Yaskawa INFORM job: SKRZYNIA_5340_-90_STOPNI_20BR.JBI

/JOB
//NAME SKRZYNIA_5340_-90_STOPNI_20BR
///FOLDERNAME 02-SKRZYNIE_JOBS
//POS
///NPOS 615,615,0,39,0,0
///TOOL 0
///POSTYPE PULSE
///PULSE
C00000=0,-52280,40443,0,6876,0
C00001=-82314,-24956,17040,-59626,-27382,-6248
C00002=-93910,-8625,17040,-59626,-43355,-6248
C00003=-98846,-1061,-42166,-80308,-57081,16120
C00004=-100452,6057,-48127,-85711,-56704,21322
C00005=-95817,31791,-34187,-84788,-63710,26674
C00006=-95573,33077,-33257,-84645,-64023,26851
C00007=-94315,33778,-32137,-85160,-63467,26714
C00008=-95573,33077,-33257,-84645,-64023,26851
C00009=-94948,31301,-36075,-85235,-63717,27152
C00010=-95573,33077,-33257,-84645,-64023,26851
C00011=-95263,33142,-33256,-84677,-63995,26850
C00012=-95263,33142,-33256,-84677,-63995,26850
C00013=-94230,33719,-32331,-85099,-63538,26735
C00014=-95263,33142,-33256,-84677,-63995,26850
C00015=-94794,31816,-35365,-85120,-63763,27076
C00016=-95263,33142,-33256,-84677,-63995,26850
C00017=-95260,33144,-33256,-84678,-63995,26850
C00018=-95260,33144,-33256,-84678,-63995,26850
C00019=-94260,33701,-32361,-85086,-63552,26738
C00020=-95260,33144,-33256,-84678,-63995,26850
C00021=-94835,31943,-35167,-85080,-63786,27056
C00022=-95260,33144,-33256,-84678,-63995,26850
C00023=-95258,25631,32269,-66559,-75499,2416
C00024=-95258,25631,32269,-66559,-75499,2416
C00025=-94256,26435,33444,-66420,-74940,2208
C00026=-95258,25631,32269,-66559,-75499,2416
C00027=-94857,24030,29962,-66606,-75105,2539
C00028=-95258,25631,32269,-66559,-75499,2416
C00029=-98811,21047,-15512,-99242,-81394,20987
C00030=-98811,21047,-15512,-99242,-81394,20987
C00031=-97856,21592,-14760,-99539,-80803,20995
C00032=-98811,21047,-15512,-99242,-81394,20987
C00033=-98487,19855,-17143,-99373,-81250,21110
C00034=-98811,21047,-15512,-99242,-81394,20987
C00035=-99077,36985,67047,-90824,-74996,11
C00036=-99077,36985,67047,-90824,-74996,11
C00037=-98126,38026,68808,-90519,-74354,-175
C00038=-99077,36985,67047,-90824,-74996,11
C00039=-98675,34279,62554,-90994,-74807,523
C00040=-99077,36985,67047,-90824,-74996,11
C00041=-98046,30065,45001,-99674,-75008,5996
C00042=-96663,27244,32711,-106417,-76052,10001
C00043=-96035,27733,33435,-106407,-75606,10011
C00044=-96663,27244,32711,-106417,-76052,10001
C00045=-96274,25568,30264,-106516,-75947,10234
C00046=-96663,27244,32711,-106417,-76052,10001
C00047=-93416,-2088,4699,-99676,-50441,9343
C00048=-88080,-20128,-3199,-80943,-31244,2335
C00049=-48287,-55439,-44481,-48508,-5390,-10469
C00050=-48287,-44591,-17414,-16172,-14532,-25809
C00051=-85348,-13130,13838,-41209,-47455,-8220
C00052=-97998,22495,32685,-69647,-75009,8900
C00053=-97362,30289,38867,-71738,-79704,10396
C00054=-97362,30289,38867,-71738,-79704,10396
C00055=-96447,31020,39967,-71637,-79179,10220
C00056=-97362,30289,38867,-71738,-79704,10396
C00057=-97069,28896,36765,-71776,-79401,10550
C00058=-97362,30289,38867,-71738,-79704,10396
C00059=-99590,25338,21334,-81459,-78469,-3358
C00060=-99590,25338,21334,-81459,-78469,-3358
C00061=-98681,25943,22203,-81468,-77867,-3455
C00062=-99590,25338,21334,-81459,-78469,-3358
C00063=-99296,24016,19444,-81525,-78239,-3225
C00064=-99590,25338,21334,-81459,-78469,-3358
C00065=-99820,26032,21623,-82067,-78848,-4447
C00066=-99820,26032,21623,-82067,-78848,-4447
C00067=-98898,26645,22513,-82083,-78237,-4546
C00068=-99820,26032,21623,-82067,-78848,-4447
C00069=-99438,24292,19129,-82156,-78552,-4268
C00070=-99820,26032,21623,-82067,-78848,-4447
C00071=-95331,1432,-9864,-84798,-60031,-3557
C00072=-95107,2197,-5510,-96695,-61306,-2364
C00073=-99461,26071,27151,-92834,-78756,-5773
C00074=-99144,26285,27462,-92832,-78536,-5787
C00075=-98121,27001,28507,-92822,-77820,-5838
C00076=-99144,26285,27462,-92832,-78536,-5787
C00077=-98815,24779,25284,-92901,-78347,-5607
C00078=-99144,26285,27462,-92832,-78536,-5787
C00079=-91210,-11403,-27677,-113165,-52408,5733
C00080=-98271,-15326,-41207,-114268,-59488,7673
C00081=-83743,-25164,-57719,-138536,-50905,17366
C00082=-83743,-25361,-52011,-136459,-47698,15842
C00083=-93071,-30029,-62286,-132724,-54351,14554
C00084=-61872,-66272,-83954,-148251,-32298,21081
C00085=-61872,-49557,-32264,-110357,-15428,1928
C00086=-65143,-26385,24751,-20080,-56896,-30933
C00087=-94996,555,46629,-41386,-61308,-21898
C00088=-98483,-26598,-36123,-71694,-41449,-2503
C00089=-98197,-8670,-25604,-81540,-55001,4479
C00090=-99236,18416,3235,-80713,-73731,6125
C00091=-98716,22747,8680,-80557,-75862,6048
C00092=-97982,23215,9333,-80619,-75386,5974
C00093=-98716,22747,8680,-80557,-75862,6048
C00094=-98409,21490,6932,-80649,-75627,6156
C00095=-98716,22747,8680,-80557,-75862,6048
C00096=-91715,3355,37300,-53415,-58440,-15905
C00097=-100183,29342,35466,-85708,-79719,1114
C00098=-100183,29342,35466,-85708,-79719,1114
C00099=-99011,30198,36753,-85631,-78926,990
C00100=-100183,29342,35466,-85708,-79719,1114
C00101=-99817,27493,32713,-85776,-79458,1347
C00102=-100183,29342,35466,-85708,-79719,1114
C00103=-99593,21150,23680,-85914,-74803,1967
C00104=-99593,30181,53843,-82632,-75568,-4688
C00105=-99618,36376,62891,-83676,-78551,-5246
C00106=-98461,37549,64848,-83362,-77827,-5489
C00107=-99618,36376,62891,-83676,-78551,-5246
C00108=-99260,34032,59054,-83761,-78261,-4840
C00109=-99618,36376,62891,-83676,-78551,-5246
C00110=-94729,-288,3800,-87543,-55904,1533
C00111=-77861,-26606,-19905,-76223,-21443,-3330
C00112=-46440,-50562,-32626,1826,-13880,-39178
C00113=-46440,-50562,-32626,1826,-13880,-39178
C00114=-38692,-65390,10180,-18335,3144,1955
C00115=0,-52280,40443,0,6876,0
C00116=0,-52280,40443,0,6876,0
C00117=0,-43112,23163,32261,-40956,29092
C00118=-48283,-21883,28214,-25170,-26491,48363
C00119=-46664,-3144,58041,-18842,-32105,45325
C00120=-50347,-18571,12268,-49104,-16423,60029
C00121=-52476,-17044,12146,-55476,-16783,62883
C00122=-51467,-16091,12918,-54586,-16145,62570
C00123=-51762,-16375,12685,-54854,-16332,62665
C00124=-53129,-15664,13268,-57063,-16995,63582
C00125=-52557,-17119,12084,-55547,-16837,62908
C00126=-52557,-17119,12084,-55547,-16837,62908
C00127=-52367,-16944,12224,-55385,-16717,62852
C00128=-50800,-15431,13458,-53958,-15729,62345
C00129=-51041,-15672,13259,-54187,-15881,62428
C00130=-52118,-15296,13570,-55899,-16415,63135
C00131=-51917,-16522,12564,-54988,-16433,62714
C00132=-50509,-19000,10610,-51503,-15997,61182
C00133=-52966,-16930,12240,-56194,-17032,63176
C00134=-51879,-15912,13067,-55265,-16346,62852
C00135=-52154,-16175,12851,-55507,-16521,62938
C00136=-53227,-15612,13314,-57215,-17042,63646
C00137=-52966,-16930,12240,-56194,-17032,63176
C00138=-50703,-18403,11066,-52155,-16024,61477
C00139=-52780,-17619,11680,-55562,-17015,62889
C00140=-51306,-16241,12790,-54268,-16084,62435
C00141=-51660,-16583,12512,-54593,-16308,62551
C00142=-53327,-15718,13220,-57282,-17114,63667
C00143=-52780,-17619,11680,-55562,-17015,62889
C00144=-50704,-18401,11069,-52157,-16021,61478
C00145=-53191,-17342,11901,-56260,-17204,63181
C00146=-51773,-16022,12969,-55050,-16305,62760
C00147=-52146,-16378,12679,-55379,-16540,62876
C00148=-53214,-15820,13135,-57085,-17059,63584
C00149=-53002,-17172,12037,-56105,-17083,63128
C00150=-51005,-17995,11387,-52847,-16122,61778
C00151=-52654,-17319,11922,-55560,-16911,62904
C00152=-51372,-16113,12897,-54432,-16099,62508
C00153=-51648,-16379,12679,-54684,-16273,62598
C00154=-52952,-15703,13233,-56807,-16903,63480
C00155=-53323,-17134,12070,-56539,-17248,63304
C00156=-52826,-20105,4812,-63938,-15678,66983
C00157=-52298,-19620,5183,-63681,-15322,66914
C00158=-51076,-18450,6096,-63049,-14499,66733
C00159=-51419,-18785,5831,-63233,-14731,66786
C00160=-52680,-18133,6347,-65138,-15424,67581
C00161=-52924,-19431,7025,-60935,-16175,65505
C00162=-51752,-18759,10786,-53484,-16613,62002
C00163=-52244,-17884,11471,-54682,-16766,62529
C00164=-50303,-16031,12961,-52880,-15542,61887
C00165=-50741,-16464,12607,-53310,-15818,62044
C00166=-52416,-15612,13306,-56135,-16617,63223
C00167=-51898,-18011,11369,-54129,-16600,62301
C00168=-50945,-18019,11363,-52741,-16103,61737
C00169=-51347,-17395,11856,-53690,-16237,62152
C00170=-49990,-16073,12923,-52376,-15383,61677
C00171=-50384,-16465,12603,-52769,-15629,61822
C00172=-52066,-15616,13298,-55654,-16423,63028
C00173=-51792,-17610,11685,-54205,-16494,62350
C00174=-50945,-18019,11363,-52741,-16103,61737
C00175=-50845,-17493,11778,-52895,-15987,61824
C00176=-49521,-16191,12826,-51571,-15155,61341
C00177=-49894,-16567,12520,-51958,-15389,61484
C00178=-51728,-15654,13268,-55171,-16246,62832
C00179=-51082,-17431,11827,-53280,-16102,61986
C00180=-50028,-23690,-6096,-22921,-31075,54538
C00181=-50346,-22995,-5584,-23393,-31002,54768
C00182=-48843,-21430,-4410,-21901,-30270,54078
C00183=-49178,-21788,-4683,-22239,-30433,54235
C00184=-50538,-21100,-4158,-23908,-30654,55032
C00185=-50252,-22811,-5450,-23315,-30936,54734
C00186=-49763,-24818,-32918,-23163,-28604,59699
C00187=-49144,-24298,-32242,-22455,-28505,59304
C00188=-47766,-22458,-30816,-21237,-27774,58615
C00189=-48099,-22913,-31171,-21534,-27949,58786
C00190=-49602,-21997,-30448,-23301,-28174,59772
C00191=-49259,-23869,-32392,-22880,-28141,59533
C00192=-50713,-12366,-58367,-41124,-17813,74400
C00193=-50097,-11438,-57505,-40749,-17495,74109
C00194=-49105,-9842,-55994,-40096,-16991,73614
C00195=-49355,-10250,-56383,-40269,-17116,73742
C00196=-50506,-9357,-55529,-41571,-17503,74586
C00197=-49771,-10920,-57018,-40545,-17327,73951
C00198=-46548,-30139,-39639,-20061,-27197,57955
C00199=-48797,-26670,-6576,-20404,-32539,53259
C00200=-45389,-28224,4312,-35967,-15579,54278
C00201=-40154,-51179,-915,-24203,-8234,36524
C00202=0,-52280,40443,0,6876,0
C00203=0,-52280,40443,0,6876,0
C00204=-2117,-50103,-33543,-4117,45077,85249
C00205=26439,-48928,-33543,-4117,-52362,85249
C00206=26439,-27355,-33543,-41485,-52362,85249
C00207=39218,-24492,-41653,-51934,-39374,86964
C00208=38244,-2284,-24157,-56964,-37300,90090
C00209=26640,586,-20198,-77712,-51919,89712
C00210=26323,460,-20341,-77681,-52125,89737
C00211=25607,3186,-17293,-77585,-52601,89760
C00212=26323,460,-20341,-77681,-52125,89737
C00213=27719,1044,-19697,-77798,-51218,89644
C00214=26640,586,-20198,-77712,-51919,89712
C00215=46457,7101,-11330,-26648,-40775,82885
C00216=47439,8350,-9833,-26106,-40556,82449
C00217=46334,10684,-6981,-26557,-41070,82837
C00218=47439,8350,-9833,-26106,-40556,82449
C00219=48354,9159,-8854,-25603,-40343,82046
C00220=47439,8350,-9833,-26106,-40556,82449
C00221=24760,-3019,-10726,-94610,-54398,89614
C00222=25145,-1220,-8811,-94681,-54143,89655
C00223=24492,1290,-6066,-94601,-54582,89624
C00224=25145,-1220,-8811,-94681,-54143,89655
C00225=26584,-669,-8211,-94866,-53174,89734
C00226=25145,-1220,-8811,-94681,-54143,89655
C00227=14532,-15164,-22494,-92943,-61192,88617
C00228=-33377,-12679,-20251,-90012,-93751,87621
C00229=-32674,-7309,22058,-70557,-98373,80594
C00230=20046,-29908,-41690,-58842,-55822,75080
C00231=46158,10269,-6164,-23128,-46470,70172
C00232=51306,10256,-19432,-23475,-33025,71236
C00233=50386,12004,-17260,-23922,-33430,71616
C00234=51306,10256,-19432,-23475,-33025,71236
C00235=51995,10928,-18601,-23012,-32906,70879
C00236=51306,10256,-19432,-23475,-33025,71236
C00237=50667,8104,-22050,-23976,-33027,71608
C00238=27434,3323,14960,-56922,-57501,78346
C00239=29014,6574,18756,-56344,-56678,77965
C00240=28326,9009,21700,-56459,-57175,78009
C00241=29014,6574,18756,-56344,-56678,77965
C00242=30292,7183,19486,-55908,-55969,77693
C00243=29014,6574,18756,-56344,-56678,77965
C00244=24457,-1296,-8898,-94600,-54606,89622
C00245=24457,-1296,-8898,-94600,-54606,89622
C00246=23939,748,-6672,-94541,-54956,89598
C00247=24457,-1296,-8898,-94600,-54606,89622
C00248=25626,-864,-8432,-94748,-53818,89684
C00249=24457,-1296,-8898,-94600,-54606,89622
C00250=22058,-20035,-26567,-93333,-56013,88551
C00251=-28907,-25632,-31027,-90338,-90583,86609
C00252=-23923,-11573,-19230,-90501,-87328,87840
C00253=-8646,-8251,-7782,-76032,-82054,83740
C00254=42001,26537,64712,-25019,-74648,68382
C00255=42692,25604,59505,-25067,-71864,68798
C00256=42100,27723,62792,-25233,-72628,68820
C00257=42692,25604,59505,-25067,-71864,68798
C00258=43179,26157,60355,-24838,-71882,68629
C00259=42692,25604,59505,-25067,-71864,68798
C00260=42064,17796,48100,-25604,-70267,69397
C00261=28113,-7386,-15136,-95790,-47335,90009
C00262=28228,-6488,-14240,-95859,-47266,90053
C00263=27767,-5044,-12775,-95858,-47588,90072
C00264=28228,-6488,-14240,-95859,-47266,90053
C00265=29468,-5989,-13737,-96077,-46438,90154
C00266=28228,-6488,-14240,-95859,-47266,90053
C00267=51937,664,-7429,-160484,-50080,89770
C00268=52345,1107,-6938,-160727,-50007,89930
C00269=51359,2767,-5080,-160136,-50147,89540
C00270=52345,1107,-6938,-160727,-50007,89930
C00271=53054,1752,-6222,-161147,-49882,90209
C00272=52345,1107,-6938,-160727,-50007,89930
C00273=51937,664,-7429,-160484,-50080,89770
C00274=29691,-10745,-18393,-95770,-46230,89933
C00275=26663,-19279,-25970,-94307,-48104,89008
C00276=29542,-7588,-14846,-100915,-46930,90773
C00277=29616,-6902,-10165,-96183,-45225,84004
C00278=29097,-5391,-8640,-96201,-45588,84023
C00279=29616,-6902,-10165,-96183,-45225,84004
C00280=31098,-6282,-9543,-96410,-44233,84135
C00281=29616,-6902,-10165,-96183,-45225,84004
C00282=7576,-30273,-44451,-97512,-61182,86443
C00283=-18624,-40022,-50597,-93591,-78329,83668
C00284=-32134,-30783,-37092,-96173,-88064,83581
C00285=23774,-1324,-8929,-94512,-55065,89585
C00286=23774,-1324,-8929,-94512,-55065,89585
C00287=23319,517,-6924,-94461,-55372,89567
C00288=23774,-1324,-8929,-94512,-55065,89585
C00289=25077,-853,-8421,-94674,-54188,89653
C00290=23774,-1324,-8929,-94512,-55065,89585
C00291=22107,-1052,28039,-94807,-51389,77849
C00292=19995,-16885,24938,-75612,-39910,62837
C00293=8393,-42921,36369,-24238,-5473,19544
C00294=0,-52280,40443,0,6876,0
C00295=-82314,-24956,17040,-59626,-27382,-6248
C00296=-93910,-8625,17040,-59626,-43355,-6248
C00297=-98846,-1061,-42166,-80308,-57081,16120
C00298=-100452,6057,-48127,-85711,-56704,21322
C00299=-95564,34698,-34234,-85516,-63941,27819
C00300=-94021,36658,-30981,-84167,-64832,27454
C00301=-93851,36773,-30815,-84181,-64812,27439
C00302=-95564,34698,-34234,-85516,-63941,27819
C00303=-96930,32282,-32252,-82595,-65816,26305
C00304=-93901,32995,-31122,-83953,-64436,26132
C00305=-93891,32978,-31150,-83961,-64431,26134
C00306=-96930,32282,-32252,-82595,-65816,26305
C00307=-97719,-4194,-31542,-76086,-54596,10626
C00308=-88377,-34186,-45291,-67238,-52212,2442
C00309=-73560,-62084,7826,-28695,-34737,-3666
C00310=0,-52280,40443,0,6876,0
C00311=0,-52280,40443,0,6876,0
C00312=-2117,-50103,-33543,-4117,45077,85249
C00313=26439,-48928,-33543,-4117,-52362,85249
C00314=26439,-27355,-33543,-41485,-52362,85249
C00315=39218,-24492,-41653,-51934,-39374,86964
C00316=37381,-5106,-22608,-53943,-39515,88347
C00317=38119,-10689,-19379,-70548,-34101,88029
C00318=37906,-14512,-22901,-69984,-34376,87713
C00319=41414,6981,-5927,-33889,-45598,86373
C00320=42289,10624,-1511,-33365,-45508,85956
C00321=42351,10656,-1473,-33340,-45486,85935
C00322=41414,6981,-5927,-33889,-45598,86373
C00323=53221,-12364,-8957,-19277,-47766,73858
C00324=11365,-15171,10010,-30164,-77975,82960
C00325=16156,-38280,11293,-23671,-42998,42040
C00326=11365,-47379,10010,-30164,3063,681
C00327=0,-52280,40443,0,6876,0
C00328=0,-36700,24612,42871,-31823,33862
C00329=-44403,-30110,7154,-24155,-23805,45557
C00330=-51570,-19542,10947,-41619,-21811,53396
C00331=-51570,-17239,16856,-38066,-23574,51584
C00332=-55052,-13712,19754,-43494,-24529,53873
C00333=-55190,-12778,21730,-42693,-25060,53437
C00334=-40431,-28773,9158,-17648,-23273,42875
C00335=0,-36700,24612,42871,-31823,33862
C00336=0,-52280,40443,0,6876,0
C00337=0,-52280,40443,0,6876,0
C00338=-73560,-62084,7826,-28695,-34737,-3666
C00339=-88377,-34186,-45291,-67238,-52212,2442
C00340=-99860,-8392,-35780,-75647,-56000,10650
C00341=-100432,21324,12575,-83706,-77956,7498
C00342=-100432,21324,12575,-83706,-77956,7498
C00343=-97477,24790,17443,-83584,-77881,7143
C00344=-97548,25214,18044,-83537,-78171,7107
C00345=-100432,21324,12575,-83706,-77956,7498
C00346=-100473,21504,12824,-83696,-77986,7482
C00347=-97708,25565,18549,-83502,-78342,7077
C00348=-97720,26100,19317,-83456,-78605,7025
C00349=-100432,21324,12575,-83706,-77956,7498
C00350=-98403,3681,-8965,-86029,-63956,7946
C00351=-98851,2841,7216,-80537,-62817,1838
C00352=-99868,-33,22146,-72719,-59601,-5126
C00353=-99028,-10516,17309,-71061,-60695,-4227
C00354=-58820,-39124,10926,-53325,-41870,-3759
C00355=0,-52280,40443,0,6876,0
C00356=-37281,-50778,-9546,-79570,-75313,71156
C00357=-21038,-23698,-30323,-82948,-81132,85647
C00358=-21230,-24252,-33397,-84866,-81311,86227
C00359=26224,-11477,-22521,-89106,-49066,87170
C00360=30473,789,4724,-68168,-47848,79016
C00361=30460,-1091,-3608,-71823,-46530,81583
C00362=26224,-11477,-22521,-89106,-49066,87170
C00363=1250,-26379,-34995,-85812,-66036,85728
C00364=-29373,-17697,-13794,-84248,-87305,82376
C00365=-12562,-22815,-22029,-52123,-75138,85349
C00366=41964,2536,-13642,-34848,-42769,74522
C00367=37974,4101,-26304,-58477,-36842,84551
C00368=37992,4823,-31618,-63468,-34913,87461
C00369=41439,5489,-14791,-37032,-40569,75962
C00370=38833,-3286,10682,-41231,-51577,69207
C00371=-9276,-22918,-17698,-90837,-69000,78700
C00372=-8172,-56778,-49528,-75726,-40055,75711
C00373=-3982,-61001,-53003,-69042,-33087,73336
C00374=37287,-55159,35520,-2191,5667,2084
C00375=0,-52280,40443,0,6876,0
C00376=0,-36700,24612,42871,-31823,33862
C00377=-44403,-30110,7154,-24155,-23805,45557
C00378=-44403,-30110,7154,-24155,-23805,45557
C00379=-42101,-12213,25656,-103795,-5192,78630
C00380=-46259,-8171,27719,-110365,-8144,81138
C00381=-49067,-3914,32085,-108223,-9817,79727
C00382=-55938,-2414,24284,-132193,-25662,89374
C00383=-55195,18277,75263,-85826,-17009,66357
C00384=-37783,26295,96734,15514,-13481,23189
C00385=-56934,-15752,2926,-132390,-27589,90381
C00386=-47073,-34549,9488,-27883,-30316,51458
C00387=0,-52280,40443,0,6876,0
C00388=0,-52280,40443,0,6876,0
C00389=-73560,-62084,7826,-28695,-34737,-3666
C00390=-96366,-17217,16860,-56620,-71703,-18245
C00391=-98152,-14905,2044,-65675,-67485,-3494
C00392=-100467,-7393,-15195,-81625,-60158,6002
C00393=-99336,18440,8642,-84276,-74234,7647
C00394=-99336,18440,8642,-84276,-74234,7647
C00395=-97907,25479,18429,-83510,-78268,7080
C00396=-97774,25771,18838,-83486,-78362,7054
C00397=-99336,18440,8642,-84276,-74234,7647
C00398=-99336,20364,19482,-82786,-74642,4774
C00399=-98337,25059,18813,-87846,-78771,10707
C00400=-98337,23926,10585,-88652,-78855,12971
C00401=-99528,19847,13673,-83665,-74506,6500
C00402=-89817,-17341,-38408,-97132,-45323,12250
C00403=-100347,-21961,-42251,-93939,-52125,11121
C00404=-60204,-59872,-73451,-117647,-17639,18840
C00405=-37721,-67612,11381,-1325,-438,-7850
C00406=0,-52280,40443,0,6876,0
C00407=37287,-55159,35520,-2191,5667,2084
C00408=40042,-68802,-18337,-47708,-19461,45384
C00409=16481,-63411,-38742,-86271,-37962,67106
C00410=28646,-23138,-32952,-89786,-42552,85395
C00411=38882,-16596,-17625,-44304,-41043,72768
C00412=40930,-6862,-13364,-47045,-37020,74415
C00413=41744,-3361,-9781,-46774,-36492,74231
C00414=41678,-4243,-16493,-50979,-33997,76666
C00415=40930,-6862,-13364,-47045,-37020,74415
C00416=38882,-16596,-17625,-44304,-41043,72768
C00417=28646,-23138,-32952,-89786,-42552,85395
C00418=29905,-15291,-26411,-91102,-43435,86304
C00419=31540,-7654,-19248,-92177,-42391,86919
C00420=31445,-8095,-22888,-97196,-43117,89457
C00421=29637,-16450,-35189,-96198,-44206,89682
C00422=-7164,-46429,-55577,-86274,-68578,84143
C00423=40042,-68802,-18337,-47708,-19461,45384
C00424=37287,-55159,35520,-2191,5667,2084
C00425=0,-52280,40443,0,6876,0
C00426=-37164,-60659,6466,-13301,-5027,19773
C00427=-45362,-39990,2831,-27538,-17767,40935
C00428=-57189,-26834,-7130,-38780,-31731,51561
C00429=-55974,-20661,-3180,-39617,-29741,52134
C00430=-55991,-28453,-45977,-64163,-20900,63765
C00431=-57189,-26834,-7130,-38780,-31731,51561
C00432=-41180,-61187,4729,-17280,-8498,23442
C00433=0,-52280,40443,0,6876,0
C00434=0,-52280,40443,0,6876,0
C00435=-43180,-50572,-20637,-6552,-29302,-38834
C00436=-79425,-37128,-15462,-51820,-35721,-18807
C00437=-93702,-21743,-5664,-65079,-41536,-12324
C00438=-94876,-11469,-23586,-124528,-59237,5423
C00439=-92861,23404,17376,-116518,-76732,-1573
C00440=-91304,28381,24747,-115873,-78046,-2652
C00441=-91460,31648,35777,-114879,-76291,-4970
C00442=-92889,23503,17516,-116511,-76737,-1586
C00443=-94876,-11469,-23586,-124528,-59237,5423
C00444=-94108,-26192,-19530,-80749,-38523,-6311
C00445=-79425,-37128,-15462,-51820,-35721,-18807
C00446=-44920,-50063,-20090,-8739,-29356,-37564
C00447=-37721,-67612,11381,-1325,-438,-7850
C00448=0,-52280,40443,0,6876,0
C00449=40043,-68802,-18337,-47706,-19461,45383
C00450=27078,-46675,7729,-35821,-60236,53359
C00451=37661,6027,34279,-36092,-58837,68690
C00452=38848,9668,32452,-36978,-55195,69693
C00453=45203,15557,41040,-24527,-60177,66840
C00454=37661,2340,23735,-37788,-55306,70200
C00455=22173,-30639,7984,-58136,-45615,60133
C00456=37287,-55159,35520,-2191,5667,2084
C00457=0,-52280,40443,0,6876,0
C00458=-23708,-46776,23536,-16027,-4787,19738
C00459=-50917,-40459,4132,-34421,-18173,42391
C00460=-54964,-26842,8528,-44141,-23181,52038
C00461=-51719,-20944,8196,-48593,-18539,54728
C00462=-53338,-16066,12564,-52314,-18938,56375
C00463=-53668,-14237,17353,-48629,-20286,54493
C00464=-18010,-41727,-5437,24633,-20435,23511
C00465=-41180,-61187,4729,-17280,-8498,23442
C00466=0,-52280,40443,0,6876,0
C00467=0,-52280,40443,0,6876,0
C00468=-37721,-67612,11381,-1325,-438,-7850
C00469=-43180,-50572,-20637,-6552,-29302,-38834
C00470=-79425,-37128,-15462,-51820,-35721,-18807
C00471=-92377,-33385,-41303,-83059,-36844,-1354
C00472=-98996,-8012,-20669,-89286,-58253,3196
C00473=-99186,-1007,-13605,-90357,-63007,3800
C00474=-99448,23410,16807,-87478,-77479,2357
C00475=-98529,24761,18725,-87324,-78429,2215
C00476=-98419,25196,20150,-87169,-78534,1864
C00477=-99450,-173,-12700,-90327,-63185,3798
C00478=-99875,3426,-9244,-98609,-66692,6315
C00479=-99431,-3293,-16601,-99643,-62713,6757
C00480=-92822,-26306,-37175,-103295,-43881,7703
C00481=-68601,-52593,-52127,-95725,-25602,3235
C00482=-80632,-38079,-20908,-64053,-45216,-12949
C00483=-43180,-50572,-20637,-6552,-29302,-38834
C00484=-37721,-67612,11381,-1325,-438,-7850
C00485=0,-52280,40443,0,6876,0
C00486=-7830,-25136,17099,-55306,-64068,52084
C00487=34592,-23156,18291,-29932,-45204,43222
C00488=27626,-5609,7480,-74303,-46810,69713
C00489=30162,-7263,-3756,-79871,-43922,73611
C00490=30945,-3557,12,-79972,-43367,73694
C00491=30934,-3652,-86,-79966,-43372,73693
C00492=29106,-7674,-4162,-79972,-44640,73655
C00493=-2837,-32019,-23857,-80741,-66785,72567
C00494=9534,-43450,13514,-26959,-29486,38723
C00495=22834,-59963,22946,-6692,-2150,9612
C00496=0,-52280,40443,0,6876,0
C00497=-23708,-46776,23536,-16027,-4787,19738
C00498=-50917,-40459,4132,-34421,-18173,42391
C00499=-51059,-36587,4608,-36647,-19418,45358
C00500=-50113,-22729,10834,-36393,-23396,50963
C00501=-58003,-17258,7975,-66354,-22196,69294
C00502=-57660,-15851,11780,-61832,-22634,66694
C00503=-50113,-22729,10834,-36393,-23396,50963
C00504=-45969,-44671,-42317,80322,10570,10889
C00505=-31285,-69981,-10849,-7246,-6842,20992
C00506=0,-52280,40443,0,6876,0
C00507=-37721,-67612,11381,-1325,-438,-7850
C00508=-43180,-50572,-20637,-6552,-29302,-38834
C00509=-79425,-37128,-15462,-51820,-35721,-18807
C00510=-92377,-33385,-41303,-83059,-36844,-1354
C00511=-97955,-4566,-17156,-86109,-58691,2381
C00512=-98023,-4368,-16953,-86108,-58737,2386
C00513=-97622,-3602,-16155,-86160,-58465,2400
C00514=-99754,24347,18348,-83049,-78046,1543
C00515=-98401,23935,17754,-83131,-77323,1564
C00516=-98274,24050,17917,-83129,-77329,1551
C00517=-99954,24418,19993,-82828,-78557,1051
C00518=-99712,24798,18984,-83012,-78332,1506
C00519=-99852,25442,19906,-82977,-78439,1439
C00520=-98294,26390,21274,-82926,-78604,1336
C00521=-98320,27540,23370,-82787,-79202,1083
C00522=-100298,21581,9800,-87114,-77804,3862
C00523=-100167,24076,23961,-91830,-78070,1153
C00524=-97934,23655,23660,-91877,-76543,1161
C00525=-97934,26645,35668,-90599,-76116,-1688
C00526=-100333,13965,-3660,-96424,-75767,7039
C00527=-99852,25442,19906,-82977,-78439,1439
C00528=-99768,8894,-2445,-89351,-68751,3793
C00529=-96099,-3787,-16815,-92200,-58195,4535
C00530=-97559,-25159,-36085,-93407,-46496,3918
C00531=-68601,-52593,-52127,-95725,-25602,3235
C00532=-80632,-38079,-20908,-64053,-45216,-12949
C00533=-43180,-50572,-20637,-6552,-29302,-38834
C00534=-37721,-67612,11381,-1325,-438,-7850
C00535=54026,-30203,28811,7745,-28969,5087
C00536=55906,-29650,27841,6704,-28568,42061
C00537=3910,-49110,-20873,-64325,-51391,71742
C00538=9596,-41005,-15480,-61992,-50741,70573
C00539=34629,-5327,8260,-51720,-47880,65426
C00540=35679,2837,17551,-51053,-47466,65038
C00541=35689,-56,7549,-54586,-44718,67469
C00542=34629,-5327,8260,-51720,-47880,65426
C00543=9596,-41005,-15480,-61992,-50741,70573
C00544=29660,-4584,-26917,-122917,-59269,85605
C00545=30458,-1431,-23593,-123278,-58903,85810
C00546=32051,-581,-21149,-126899,-58917,85995
C00547=28378,-5181,-30467,-124970,-61925,86269
C00548=9596,-41005,-15480,-61992,-50741,70573
C00549=4124,-42500,-16101,-63937,-54198,71061
C00550=22834,-59963,22946,-6692,-2150,9612
C00551=0,-52280,40443,0,6876,0
C00552=-44101,-76445,-48847,-15697,-17168,40457
C00553=-48984,-30078,-36716,-21434,-29637,58750
C00554=-50484,-13386,-55713,-36158,-19724,71897
C00555=-50319,-9878,-52358,-36554,-19395,72071
C00556=-57778,15231,-57159,-77377,-21293,89265
C00557=-50484,-13386,-55713,-36158,-19724,71897
C00558=-49763,-25421,-36239,-24565,-26935,60445
C00559=-50529,-22709,-3778,-22940,-31995,54502
C00560=-45389,-28224,4312,-35967,-15579,54278
C00561=-40154,-51179,-915,-24203,-8234,36524
C00562=0,-52280,40443,0,6876,0
C00563=0,-52280,40443,0,6876,0
C00564=-37721,-67612,11381,-1325,-438,-7850
C00565=-43180,-50572,-20637,-6552,-29302,-38834
C00566=-43180,-50572,-20637,-6552,-29302,-38834
C00567=-91571,-17240,10754,-52986,-45776,-17944
C00568=-95322,4002,18806,-71534,-58652,-8117
C00569=-84901,-1641,24348,-52361,-47087,-17020
C00570=-100018,24469,26124,-84922,-77496,-993
C00571=-98221,24171,26084,-84881,-76275,-1110
C00572=-97925,23780,23736,-81145,-76027,-1196
C00573=-96763,24072,23316,-74311,-75270,-2269
C00574=-95281,25990,27886,-68316,-75415,-4201
C00575=-99355,23812,23162,-76774,-76908,-1703
C00576=-99772,22813,18672,-85812,-76963,849
C00577=-98588,26860,21106,-87462,-79585,-1754
C00578=-98621,27173,20618,-87985,-79896,-2348
C00579=-99360,20896,24116,-84704,-74336,-1671
C00580=-99329,20456,17173,-93067,-75506,1686
C00581=-97621,19686,17216,-93018,-74287,1457
C00582=-97553,22128,27761,-91636,-73750,-1130
C00583=-97912,34558,59975,-88815,-75536,-7324
C00584=-97912,45071,86162,-86500,-75470,-12145
C00585=-89794,-9992,-7341,-81590,-44258,-3681
C00586=-98228,-14972,-11291,-81392,-49231,-4002
C00587=-98228,-7428,13566,-72439,-51372,-10695
C00588=-68865,-35989,-5252,-49829,-38105,-21179
C00589=-15566,-52364,-9989,12732,-35649,-46896
C00590=0,-52278,40443,-31822,-65283,46097
C00591=7820,3000,44222,-77356,-66876,70486
C00592=23103,22769,71034,-65639,-61603,67373
C00593=25078,30713,84198,-63240,-61811,65668
C00594=25008,30264,83410,-63369,-61766,65773
C00595=23103,22769,71034,-65639,-61603,67373
C00596=23103,22769,71034,-65639,-61603,67373
C00597=25078,30713,84198,-63240,-61811,65668
C00598=25008,30264,83410,-63369,-61766,65773
C00599=23103,22769,71034,-65639,-61603,67373
C00600=-3014,-20441,-7349,-104591,-68614,79454
C00601=-3014,-20441,-7349,-104591,-68614,79454
C00602=-13238,-21720,-1359,-93359,-59492,72612
C00603=10261,-46634,14475,-36899,-22136,31570
C00604=22834,-59963,22946,-6692,-2150,9612
C00605=0,-52280,40443,0,6876,0
C00606=-23708,-46776,23536,-16027,-4787,19738
C00607=-50917,-40459,4132,-34421,-18173,42391
C00608=-49876,-21948,7530,-68838,-10324,59148
C00609=-46721,-18942,9765,-68167,-8197,59205
C00610=-47734,-15041,12007,-78406,-8476,63945
C00611=-48173,-14749,12492,-78097,-8776,63748
C00612=-42573,-24036,4541,-56448,-5917,54155
C00613=-31287,-69981,-10850,-7253,-6843,20996
C00614=0,-52280,40443,0,6876,0
BC00000=455888
BC00001=445130
BC00002=445130
BC00003=445130
BC00004=445130
BC00005=467179
BC00006=468227
BC00007=468227
BC00008=468227
BC00009=468227
BC00010=468227
BC00011=514421
BC00012=514421
BC00013=514421
BC00014=514421
BC00015=514421
BC00016=514421
BC00017=560588
BC00018=560588
BC00019=560588
BC00020=560588
BC00021=560588
BC00022=560588
BC00023=536404
BC00024=536404
BC00025=536404
BC00026=536404
BC00027=536404
BC00028=536404
BC00029=582458
BC00030=582458
BC00031=582458
BC00032=582458
BC00033=582458
BC00034=582458
BC00035=581206
BC00036=581206
BC00037=581206
BC00038=581206
BC00039=581206
BC00040=581206
BC00041=608443
BC00042=626741
BC00043=626741
BC00044=626741
BC00045=626741
BC00046=626741
BC00047=604255
BC00048=604255
BC00049=627238
BC00050=699121
BC00051=714117
BC00052=772491
BC00053=770398
BC00054=770398
BC00055=770398
BC00056=770398
BC00057=770398
BC00058=770398
BC00059=820815
BC00060=820815
BC00061=820815
BC00062=820815
BC00063=820815
BC00064=820815
BC00065=866263
BC00066=866263
BC00067=866263
BC00068=866263
BC00069=866263
BC00070=866263
BC00071=866263
BC00072=904896
BC00073=904896
BC00074=904896
BC00075=904896
BC00076=904896
BC00077=904896
BC00078=904896
BC00079=872244
BC00080=872244
BC00081=872244
BC00082=872244
BC00083=872244
BC00084=872244
BC00085=872244
BC00086=943472
BC00087=944390
BC00088=976590
BC00089=976703
BC00090=960530
BC00091=953739
BC00092=953739
BC00093=953739
BC00094=953739
BC00095=953739
BC00096=949233
BC00097=963886
BC00098=963886
BC00099=963886
BC00100=963886
BC00101=963886
BC00102=963886
BC00103=963886
BC00104=1017492
BC00105=1017492
BC00106=1017492
BC00107=1017492
BC00108=1017492
BC00109=1017492
BC00110=969716
BC00111=953277
BC00112=956863
BC00113=935999
BC00114=860772
BC00115=811795
BC00116=811793
BC00117=811795
BC00118=919701
BC00119=919701
BC00120=949003
BC00121=953382
BC00122=953382
BC00123=953382
BC00124=953382
BC00125=953382
BC00126=1005542
BC00127=1006846
BC00128=1006846
BC00129=1006846
BC00130=1006846
BC00131=1006846
BC00132=888056
BC00133=888056
BC00134=888056
BC00135=888056
BC00136=888056
BC00137=888056
BC00138=830714
BC00139=830714
BC00140=830714
BC00141=830714
BC00142=830714
BC00143=830714
BC00144=764829
BC00145=764829
BC00146=764829
BC00147=764829
BC00148=764829
BC00149=764829
BC00150=707174
BC00151=707174
BC00152=707174
BC00153=707174
BC00154=707174
BC00155=707174
BC00156=642071
BC00157=642071
BC00158=642071
BC00159=642071
BC00160=642071
BC00161=642071
BC00162=584746
BC00163=584746
BC00164=584746
BC00165=584746
BC00166=584746
BC00167=584746
BC00168=519232
BC00169=519232
BC00170=519232
BC00171=519232
BC00172=519232
BC00173=519232
BC00174=461813
BC00175=461813
BC00176=461813
BC00177=461813
BC00178=461813
BC00179=461813
BC00180=459544
BC00181=459544
BC00182=459544
BC00183=459544
BC00184=459544
BC00185=459544
BC00186=459544
BC00187=459544
BC00188=459544
BC00189=459544
BC00190=459544
BC00191=459544
BC00192=459544
BC00193=459544
BC00194=459544
BC00195=459544
BC00196=459544
BC00197=459544
BC00198=459544
BC00199=459544
BC00200=459540
BC00201=533216
BC00202=533216
BC00203=492150
BC00204=423885
BC00205=423885
BC00206=423885
BC00207=423885
BC00208=423885
BC00209=423882
BC00210=423882
BC00211=423882
BC00212=423882
BC00213=423882
BC00214=423882
BC00215=517447
BC00216=516208
BC00217=516208
BC00218=516208
BC00219=516208
BC00220=516208
BC00221=462401
BC00222=462401
BC00223=462401
BC00224=462401
BC00225=462401
BC00226=462401
BC00227=462401
BC00228=462401
BC00229=581968
BC00230=647467
BC00231=647467
BC00232=647467
BC00233=647467
BC00234=647467
BC00235=647467
BC00236=647467
BC00237=647467
BC00238=600589
BC00239=600589
BC00240=600589
BC00241=600589
BC00242=600589
BC00243=600589
BC00244=646713
BC00245=646713
BC00246=646713
BC00247=646713
BC00248=646713
BC00249=646713
BC00250=646713
BC00251=646713
BC00252=703926
BC00253=764819
BC00254=734650
BC00255=734650
BC00256=734650
BC00257=734650
BC00258=734650
BC00259=734650
BC00260=734650
BC00261=762000
BC00262=762000
BC00263=762000
BC00264=762000
BC00265=762000
BC00266=762000
BC00267=768744
BC00268=768744
BC00269=768744
BC00270=768744
BC00271=768744
BC00272=768744
BC00273=768744
BC00274=762000
BC00275=762000
BC00276=869424
BC00277=869424
BC00278=869424
BC00279=869424
BC00280=869424
BC00281=869424
BC00282=869424
BC00283=869424
BC00284=983898
BC00285=992364
BC00286=992364
BC00287=992364
BC00288=992364
BC00289=992364
BC00290=992364
BC00291=927243
BC00292=910363
BC00293=791398
BC00294=458496
BC00295=445130
BC00296=445130
BC00297=445130
BC00298=445130
BC00299=475938
BC00300=475917
BC00301=468314
BC00302=475938
BC00303=515329
BC00304=515329
BC00305=508301
BC00306=515329
BC00307=542207
BC00308=542207
BC00309=542207
BC00310=542207
BC00311=492150
BC00312=423885
BC00313=423885
BC00314=423885
BC00315=423885
BC00316=418215
BC00317=406365
BC00318=406365
BC00319=507950
BC00320=507950
BC00321=500226
BC00322=507950
BC00323=493160
BC00324=493160
BC00325=493160
BC00326=493160
BC00327=493160
BC00328=582810
BC00329=655182
BC00330=714528
BC00331=712780
BC00332=712780
BC00333=773753
BC00334=773753
BC00335=582810
BC00336=540924
BC00337=542207
BC00338=542207
BC00339=542207
BC00340=590944
BC00341=543764
BC00342=459277
BC00343=459277
BC00344=451665
BC00345=459277
BC00346=520748
BC00347=520748
BC00348=528295
BC00349=520748
BC00350=524597
BC00351=612873
BC00352=584417
BC00353=584417
BC00354=584417
BC00355=584417
BC00356=542360
BC00357=599440
BC00358=482963
BC00359=482963
BC00360=482963
BC00361=482963
BC00362=482963
BC00363=482963
BC00364=482963
BC00365=633179
BC00366=633182
BC00367=633182
BC00368=633182
BC00369=633182
BC00370=590162
BC00371=577838
BC00372=565789
BC00373=612529
BC00374=620193
BC00375=620193
BC00376=812803
BC00377=887783
BC00378=927066
BC00379=893694
BC00380=914884
BC00381=914884
BC00382=943670
BC00383=952070
BC00384=963270
BC00385=945981
BC00386=853059
BC00387=542207
BC00388=542207
BC00389=513519
BC00390=556866
BC00391=576802
BC00392=590944
BC00393=571989
BC00394=566860
BC00395=566866
BC00396=572997
BC00397=566860
BC00398=625806
BC00399=632891
BC00400=631419
BC00401=627770
BC00402=635118
BC00403=635118
BC00404=633159
BC00405=733103
BC00406=733103
BC00407=620193
BC00408=620193
BC00409=625652
BC00410=635598
BC00411=635598
BC00412=635598
BC00413=635598
BC00414=635598
BC00415=635598
BC00416=635598
BC00417=635598
BC00418=658627
BC00419=658630
BC00420=665879
BC00421=658627
BC00422=658627
BC00423=620193
BC00424=620193
BC00425=620193
BC00426=561542
BC00427=498768
BC00428=452071
BC00429=452071
BC00430=452071
BC00431=452071
BC00432=524165
BC00433=524165
BC00434=733103
BC00435=733103
BC00436=615417
BC00437=615411
BC00438=615411
BC00439=615411
BC00440=615411
BC00441=615411
BC00442=615411
BC00443=615411
BC00444=615411
BC00445=615417
BC00446=698572
BC00447=733103
BC00448=733103
BC00449=667407
BC00450=721208
BC00451=721208
BC00452=721208
BC00453=727232
BC00454=730010
BC00455=686453
BC00456=620193
BC00457=620193
BC00458=576077
BC00459=541793
BC00460=580754
BC00461=589556
BC00462=589433
BC00463=647350
BC00464=649294
BC00465=561088
BC00466=547800
BC00467=733103
BC00468=733103
BC00469=733103
BC00470=733103
BC00471=757807
BC00472=750752
BC00473=747214
BC00474=740531
BC00475=740531
BC00476=745553
BC00477=740531
BC00478=750469
BC00479=750469
BC00480=750469
BC00481=750469
BC00482=783373
BC00483=795297
BC00484=733103
BC00485=733103
BC00486=727492
BC00487=727492
BC00488=759331
BC00489=759331
BC00490=759331
BC00491=766564
BC00492=759331
BC00493=759331
BC00494=672725
BC00495=672725
BC00496=672725
BC00497=766882
BC00498=791101
BC00499=802867
BC00500=836517
BC00501=836517
BC00502=895002
BC00503=836517
BC00504=798026
BC00505=767805
BC00506=733103
BC00507=733103
BC00508=733103
BC00509=733103
BC00510=768965
BC00511=777113
BC00512=815683
BC00513=817504
BC00514=817504
BC00515=817504
BC00516=824335
BC00517=824335
BC00518=862603
BC00519=862905
BC00520=863393
BC00521=870426
BC00522=870426
BC00523=904292
BC00524=904292
BC00525=904292
BC00526=904292
BC00527=862905
BC00528=824848
BC00529=818776
BC00530=812035
BC00531=750469
BC00532=783373
BC00533=795297
BC00534=733103
BC00535=762701
BC00536=765633
BC00537=830967
BC00538=835024
BC00539=852883
BC00540=852883
BC00541=852883
BC00542=852883
BC00543=835024
BC00544=861491
BC00545=861491
BC00546=861491
BC00547=861491
BC00548=835024
BC00549=835024
BC00550=672725
BC00551=672725
BC00552=528256
BC00553=459544
BC00554=459544
BC00555=459544
BC00556=459544
BC00557=459544
BC00558=459544
BC00559=459544
BC00560=459540
BC00561=533216
BC00562=533216
BC00563=733103
BC00564=733103
BC00565=854587
BC00566=967109
BC00567=948121
BC00568=961016
BC00569=923671
BC00570=946274
BC00571=946274
BC00572=946274
BC00573=946274
BC00574=946274
BC00575=946274
BC00576=970029
BC00577=970060
BC00578=977448
BC00579=970029
BC00580=1018114
BC00581=1018114
BC00582=1018114
BC00583=1018114
BC00584=1018114
BC00585=975782
BC00586=976838
BC00587=956699
BC00588=952322
BC00589=952322
BC00590=921533
BC00591=921533
BC00592=946591
BC00593=946591
BC00594=953713
BC00595=946591
BC00596=997282
BC00597=997282
BC00598=1004404
BC00599=997282
BC00600=1013986
BC00601=963295
BC00602=908449
BC00603=754884
BC00604=672725
BC00605=672725
BC00606=562340
BC00607=452362
BC00608=452362
BC00609=452362
BC00610=452362
BC00611=512870
BC00612=511886
BC00613=742282
BC00614=742282
///POSTYPE BASE
///RECTAN
///RCONF 1,0,0,0,0,0,0,0,0,0,0,0,0,0,0,0,0,0,0,0,0,0,0,0
P00006=0.000,0.000,0.000,0.0000,0.0000,0.0000
P00300=-0.036,-1.505,2.318,0.0000,0.0000,0.0000
P00301=0.046,-2.112,7.779,0.0000,0.0000,0.0000
P00302=-0.180,-2.409,6.326,0.0000,0.0000,0.0000
///RCONF 0,0,0,0,0,0,0,0,0,0,0,0,0,0,0,0,0,0,0,0,0,0,0,0
P00303=-0.004,-1.437,-4.584,0.0000,0.0000,0.0000
P00304=0.028,-1.666,-4.234,0.0000,0.0000,0.0000
P00305=-0.003,-1.920,-3.501,0.0000,0.0000,0.0000
P00306=0.015,-2.252,-3.054,0.0000,0.0000,0.0000
P00307=0.019,-2.151,-5.077,0.0000,0.0000,0.0000
P00308=-0.003,-2.092,-4.888,0.0000,0.0000,0.0000
P00309=-0.040,-2.205,-4.992,0.0000,0.0000,0.0000
P00310=-0.006,-2.490,-5.925,0.0000,0.0000,0.0000
P00311=-0.007,-2.079,-5.307,0.0000,0.0000,0.0000
P00312=-0.032,2.202,-7.632,0.0000,0.0000,0.0000
///RCONF 1,0,0,0,0,0,0,0,0,0,0,0,0,0,0,0,0,0,0,0,0,0,0,0
P00349=0.060,0.167,-1.133,0.0000,0.0000,0.0000
///RCONF 0,0,0,0,0,0,0,0,0,0,0,0,0,0,0,0,0,0,0,0,0,0,0,0
P00350=11.519,-0.008,1.149,0.0000,0.0000,0.0000
P00351=13.563,-0.027,-0.653,0.0000,0.0000,0.0000
P00352=13.252,-0.027,-0.827,0.0000,0.0000,0.0000
P00353=10.971,-0.082,0.776,0.0000,0.0000,0.0000
P00354=-0.024,2.508,-1.824,0.0000,0.0000,0.0000
P00355=-0.001,2.528,-1.131,0.0000,0.0000,0.0000
P00356=-0.034,2.921,-0.262,0.0000,0.0000,0.0000
P00357=0.003,3.386,-0.091,0.0000,0.0000,0.0000
P00358=0.014,3.037,-0.020,0.0000,0.0000,0.0000
P00359=-0.005,2.731,0.912,0.0000,0.0000,0.0000
P00360=-0.011,3.412,0.438,0.0000,0.0000,0.0000
P00361=0.018,3.050,1.253,0.0000,0.0000,0.0000
P00400=5.920,-3.503,-0.024,0.0000,0.0000,0.0000
P00401=3.430,-0.021,1.131,0.0000,0.0000,0.0000
P00402=-0.253,1.107,3.062,0.0000,0.0000,0.0000
P00403=-3.666,-0.015,5.328,0.0000,0.0000,0.0000
///RCONF 1,0,0,0,0,0,0,0,0,0,0,0,0,0,0,0,0,0,0,0,0,0,0,0
P00404=0.029,4.189,-1.030,0.0000,0.0000,0.0000
///RCONF 0,0,0,0,0,0,0,0,0,0,0,0,0,0,0,0,0,0,0,0,0,0,0,0
P00405=2.420,0.007,1.427,0.0000,0.0000,0.0000
P00406=3.513,-0.022,0.429,0.0000,0.0000,0.0000
///RCONF 1,0,0,0,1,0,0,0,0,0,0,0,0,0,0,0,0,0,0,0,0,0,0,0
P00407=-0.029,2.348,-1.469,0.0000,0.0000,0.0000
P00408=0.010,1.346,-1.479,0.0000,0.0000,0.0000
///RCONF 1,0,0,0,0,0,0,0,0,0,0,0,0,0,0,0,0,0,0,0,0,0,0,0
P00409=-0.026,2.090,-1.483,0.0000,0.0000,0.0000
P00410=0.001,4.491,-0.583,0.0000,0.0000,0.0000
///RCONF 1,0,0,0,1,0,0,0,0,0,0,0,0,0,0,0,0,0,0,0,0,0,0,0
P00411=-0.015,3.627,0.872,0.0000,0.0000,0.0000
//INST
///DATE 2024/10/28 16:55
///ATTR SC,RW
///GROUP1 RB1,BS1
NOP
CALL JOB:MOVE_INTO_TUNNEL
MOVJ C00000 BC00000 VJ=30.00
MOVJ C00001 BC00001 VJ=30.00
MOVJ C00002 BC00002 VJ=30.00
MOVL C00003 BC00003 V=500.0
MOVJ C00004 BC00004 VJ=20.00
'------------------------
'W65.3
SFTOF
'------------------------
MOVL C00005 BC00005 V=333.3
MOVL C00006 BC00006 V=166.7 PL=0
REFP 3 C00007 BC00007
CALL JOB:SEARCH-R1
SET P0300 P0006
SFTON P0300
MOVL C00008 BC00008 V=66.7 PL=0
REFP 3 C00009 BC00009
CALL JOB:SEARCH-R1
SET P0300 P0006
SFTON P0300
MOVL C00010 BC00010 V=66.7 PL=0
SFTOF
'------------------------
'W65.5
'------------------------
MOVL C00011 BC00011 V=500.0
MOVL C00012 BC00012 V=166.7 PL=0
REFP 3 C00013 BC00013
CALL JOB:SEARCH-R1
SET P0301 P0006
SFTON P0301
MOVL C00014 BC00014 V=166.7 PL=0
REFP 3 C00015 BC00015
CALL JOB:SEARCH-R1
SET P0301 P0006
SFTON P0301
MOVL C00016 BC00016 V=166.7 PL=0
SFTOF
'------------------------
'W65.7
'------------------------
MOVL C00017 BC00017 V=500.0
MOVL C00018 BC00018 V=166.7 PL=0
REFP 3 C00019 BC00019
CALL JOB:SEARCH-R1
SET P0302 P0006
SFTON P0302
MOVL C00020 BC00020 V=166.7 PL=0
REFP 3 C00021 BC00021
CALL JOB:SEARCH-R1
SET P0302 P0006
SFTON P0302
MOVL C00022 BC00022 V=166.7 PL=0
SFTOF
'------------------------
'W65.10
'------------------------
MOVL C00023 BC00023 V=500.0
MOVL C00024 BC00024 V=166.7 PL=0
REFP 3 C00025 BC00025
CALL JOB:SEARCH-R1
SET P0303 P0006
SFTON P0303
MOVL C00026 BC00026 V=166.7 PL=0
REFP 3 C00027 BC00027
CALL JOB:SEARCH-R1
SET P0303 P0006
SFTON P0303
MOVL C00028 BC00028 V=166.7 PL=0
SFTOF
'------------------------
'W65.12
'------------------------
MOVL C00029 BC00029 V=500.0
MOVL C00030 BC00030 V=166.7 PL=0
REFP 3 C00031 BC00031
CALL JOB:SEARCH-R1
SET P0304 P0006
SFTON P0304
MOVL C00032 BC00032 V=166.7 PL=0
REFP 3 C00033 BC00033
CALL JOB:SEARCH-R1
SET P0304 P0006
SFTON P0304
MOVL C00034 BC00034 V=166.7 PL=0
SFTOF
'------------------------
'W65.15
'------------------------
MOVL C00035 BC00035 V=333.3
MOVL C00036 BC00036 V=166.7 PL=0
REFP 3 C00037 BC00037
CALL JOB:SEARCH-R1
SET P0305 P0006
SFTON P0305
MOVL C00038 BC00038 V=166.7 PL=0
REFP 3 C00039 BC00039
CALL JOB:SEARCH-R1
SET P0305 P0006
SFTON P0305
MOVL C00040 BC00040 V=166.7 PL=0
SFTOF
'------------------------
'W65.17
'------------------------
MOVL C00041 BC00041 V=333.3
MOVL C00042 BC00042 V=166.7 PL=0
REFP 3 C00043 BC00043
CALL JOB:SEARCH-R1
SET P0306 P0006
SFTON P0306
MOVL C00044 BC00044 V=166.7 PL=0
REFP 3 C00045 BC00045
CALL JOB:SEARCH-R1
SET P0306 P0006
SFTON P0306
MOVL C00046 BC00046 V=166.7 PL=0
SFTOF
MOVL C00047 BC00047 V=333.3
MOVL C00048 BC00048 V=500.0
MOVL C00049 BC00049 V=500.0
MOVJ C00050 BC00050 VJ=50.00
MOVL C00051 BC00051 V=500.0
MOVL C00052 BC00052 V=500.0
'------------------------
'W65.20
'------------------------
MOVL C00053 BC00053 V=166.7
MOVL C00054 BC00054 V=166.7 PL=0
REFP 3 C00055 BC00055
CALL JOB:SEARCH-R1
SET P0307 P0006
SFTON P0307
MOVL C00056 BC00056 V=166.7 PL=0
REFP 3 C00057 BC00057
CALL JOB:SEARCH-R1
SET P0307 P0006
SFTON P0307
MOVL C00058 BC00058 V=166.7 PL=0
SFTOF
'------------------------
'W65.23
'------------------------
MOVL C00059 BC00059 V=333.3
MOVL C00060 BC00060 V=166.7 PL=0
REFP 3 C00061 BC00061
CALL JOB:SEARCH-R1
SET P0308 P0006
SFTON P0308
MOVL C00062 BC00062 V=166.7 PL=0
REFP 3 C00063 BC00063
CALL JOB:SEARCH-R1
SET P0308 P0006
SFTON P0308
MOVL C00064 BC00064 V=166.7 PL=0
SFTOF
'------------------------
'W65.25
'------------------------
MOVL C00065 BC00065 V=500.0
MOVL C00066 BC00066 V=166.7 PL=0
REFP 3 C00067 BC00067
CALL JOB:SEARCH-R1
SET P0309 P0006
SFTON P0309
MOVL C00068 BC00068 V=166.7 PL=0
REFP 3 C00069 BC00069
CALL JOB:SEARCH-R1
SET P0309 P0006
SFTON P0309
MOVL C00070 BC00070 V=166.7 PL=0
SFTOF
MOVL C00071 BC00071 V=166.7
MOVL C00072 BC00072 V=666.7
MOVL C00073 BC00073 V=166.7
MOVL C00074 BC00074 V=166.7 PL=0
REFP 3 C00075 BC00075
CALL JOB:SEARCH-R1
SET P0310 P0006
SFTON P0310
MOVL C00076 BC00076 V=166.7 PL=0
REFP 3 C00077 BC00077
CALL JOB:SEARCH-R1
SET P0310 P0006
SFTON P0310
MOVL C00078 BC00078 V=166.7 PL=0
SFTOF
MOVL C00079 BC00079 V=666.7
MOVL C00080 BC00080 V=666.7
MOVL C00081 BC00081 V=666.7
MOVL C00082 BC00082 V=666.7
MOVL C00083 BC00083 V=666.7
MOVL C00084 BC00084 V=666.7
MOVL C00085 BC00085 V=666.7
MOVL C00086 BC00086 V=666.7
MOVL C00087 BC00087 V=666.7
COMM MOVL C00088 BC00088 V=666.7
COMM MOVL C00089 BC00089 V=500.0
COMM MOVL C00090 BC00090 V=333.3
COMM '------------------------
COMM 'W65.28
COMM '------------------------
COMM MOVL C00091 BC00091 V=166.7 PL=0
COMM REFP 3 C00092 BC00092
COMM CALL JOB:SEARCH-R1
COMM SET P0310 P0006
COMM SFTON P0310
COMM MOVL C00093 BC00093 V=166.7 PL=0
COMM REFP 3 C00094 BC00094
COMM CALL JOB:SEARCH-R1
COMM SET P0310 P0006
COMM SFTON P0310
COMM MOVL C00095 BC00095 V=166.7 PL=0
COMM SFTOF
'------------------------
'W65.30
MOVL C00096 BC00096 V=166.7
'------------------------
MOVL C00097 BC00097 V=500.0
MOVL C00098 BC00098 V=166.7 PL=0
REFP 3 C00099 BC00099
CALL JOB:SEARCH-R1
SET P0311 P0006
SFTON P0311
MOVL C00100 BC00100 V=166.7 PL=0
REFP 3 C00101 BC00101
CALL JOB:SEARCH-R1
SET P0311 P0006
SFTON P0311
MOVL C00102 BC00102 V=166.7 PL=0
SFTOF
MOVL C00103 BC00103 V=166.7
MOVL C00104 BC00104 V=500.0
MOVL C00105 BC00105 V=166.7 PL=0
REFP 3 C00106 BC00106
CALL JOB:SEARCH-R1
SET P0312 P0006
SFTON P0312
MOVL C00107 BC00107 V=166.7 PL=0
REFP 3 C00108 BC00108
CALL JOB:SEARCH-R1
SET P0312 P0006
SFTON P0312
MOVL C00109 BC00109 V=166.7 PL=0
SFTOF
MOVL C00110 BC00110 V=333.3
MOVL C00111 BC00111 V=333.3
MOVL C00112 BC00112 V=333.3
MOVL C00113 BC00113 V=666.7
MOVJ C00114 BC00114 VJ=50.00
MOVJ C00115 BC00115 VJ=50.00
MOVJ C00116 BC00116 VJ=10.00
MOVJ C00117 BC00117 VJ=50.00
MOVJ C00118 BC00118 VJ=30.00
MOVJ C00119 BC00119 VJ=30.00
MOVL C00120 BC00120 V=333.3
SFTOF
'------------------------
'W251A
'------------------------
MOVL C00121 BC00121 V=166.7 PL=0
REFP 3 C00122 BC00122
CALL JOB:SEARCH-R1
SET P0350 P0006
SFTON P0350
MOVL C00123 BC00123 V=166.7 PL=0
REFP 3 C00124 BC00124
CALL JOB:SEARCH-R1
SET P0350 P0006
SFTON P0350
MOVL C00125 BC00125 V=166.7 PL=0
SFTOF
'------------------------
'W254A P
'------------------------
MOVL C00126 BC00126 V=500.0
MOVL C00127 BC00127 V=166.7 PL=0
REFP 3 C00128 BC00128
CALL JOB:SEARCH-R1
SET P0349 P0006
SFTON P0349
MOVL C00129 BC00129 V=166.7 PL=0
REFP 3 C00130 BC00130
CALL JOB:SEARCH-R1
SET P0349 P0006
SFTON P0349
MOVL C00131 BC00131 V=166.7 PL=0
SFTOF
MOVJ C00132 BC00132 VJ=40.00
MOVL C00133 BC00133 V=166.7 PL=0
REFP 3 C00134 BC00134
CALL JOB:SEARCH-R1
SET P0351 P0006
SFTON P0351
MOVL C00135 BC00135 V=166.7 PL=0
REFP 3 C00136 BC00136
CALL JOB:SEARCH-R1
SET P0351 P0006
SFTON P0351
MOVL C00137 BC00137 V=166.7 PL=0
SFTOF
'------------------------
'W254A L
'------------------------
MOVJ C00138 BC00138 VJ=40.00
MOVL C00139 BC00139 V=166.7 PL=0
REFP 3 C00140 BC00140
CALL JOB:SEARCH-R1
SET P0352 P0006
SFTON P0352
MOVL C00141 BC00141 V=166.7 PL=0
REFP 3 C00142 BC00142
CALL JOB:SEARCH-R1
SET P0352 P0006
SFTON P0352
MOVL C00143 BC00143 V=166.7 PL=0
SFTOF
'------------------------
'W250A P
'------------------------
MOVJ C00144 BC00144 VJ=40.00
MOVL C00145 BC00145 V=166.7 PL=0
REFP 3 C00146 BC00146
CALL JOB:SEARCH-R1
SET P0353 P0006
SFTON P0353
MOVL C00147 BC00147 V=66.7 PL=0
REFP 3 C00148 BC00148
CALL JOB:SEARCH-R1
SET P0353 P0006
SFTON P0353
MOVL C00149 BC00149 V=66.7 PL=0
SFTOF
'------------------------
'W250A L
'------------------------
MOVJ C00150 BC00150 VJ=40.00
MOVL C00151 BC00151 V=166.7 PL=0
REFP 3 C00152 BC00152
CALL JOB:SEARCH-R1
SET P0354 P0006
SFTON P0354
MOVL C00153 BC00153 V=66.7 PL=0
REFP 3 C00154 BC00154
CALL JOB:SEARCH-R1
SET P0354 P0006
SFTON P0354
MOVL C00155 BC00155 V=166.7 PL=0
SFTOF
'------------------------
'W253A P
'------------------------
MOVJ C00156 BC00156 VJ=40.00
MOVL C00157 BC00157 V=166.7 PL=0
REFP 3 C00158 BC00158
CALL JOB:SEARCH-R1
SET P0355 P0006
SFTON P0355
MOVL C00159 BC00159 V=166.7 PL=0
REFP 3 C00160 BC00160
CALL JOB:SEARCH-R1
SET P0355 P0006
SFTON P0355
MOVL C00161 BC00161 V=166.7 PL=0
SFTOF
'------------------------
'W253A L
'------------------------
MOVJ C00162 BC00162 VJ=40.00
MOVL C00163 BC00163 V=166.7 PL=0
REFP 3 C00164 BC00164
CALL JOB:SEARCH-R1
SET P0356 P0006
SFTON P0356
MOVL C00165 BC00165 V=166.7 PL=0
REFP 3 C00166 BC00166
CALL JOB:SEARCH-R1
SET P0356 P0006
SFTON P0356
MOVL C00167 BC00167 V=166.7 PL=0
SFTOF
'------------------------
'W256A P
'------------------------
MOVJ C00168 BC00168 VJ=40.00
MOVL C00169 BC00169 V=166.7 PL=0
REFP 3 C00170 BC00170
CALL JOB:SEARCH-R1
SET P0357 P0006
SFTON P0357
MOVL C00171 BC00171 V=166.7 PL=0
REFP 3 C00172 BC00172
CALL JOB:SEARCH-R1
SET P0357 P0006
SFTON P0357
MOVL C00173 BC00173 V=166.7 PL=0
SFTOF
'------------------------
'W256A L
'------------------------
MOVJ C00174 BC00174 VJ=40.00
MOVL C00175 BC00175 V=166.7 PL=0
REFP 3 C00176 BC00176
CALL JOB:SEARCH-R1
SET P0358 P0006
SFTON P0358
MOVL C00177 BC00177 V=166.7 PL=0
REFP 3 C00178 BC00178
CALL JOB:SEARCH-R1
SET P0358 P0006
SFTON P0358
MOVL C00179 BC00179 V=166.7 PL=0
SFTOF
'------------------------
'W252A P
'------------------------
MOVL C00180 BC00180 V=666.7
MOVL C00181 BC00181 V=166.7 PL=0
REFP 3 C00182 BC00182
CALL JOB:SEARCH-R1
SET P0359 P0006
SFTON P0359
MOVL C00183 BC00183 V=166.7 PL=0
REFP 3 C00184 BC00184
CALL JOB:SEARCH-R1
SET P0359 P0006
SFTON P0359
MOVL C00185 BC00185 V=166.7 PL=0
SFTOF
'------------------------
'W252A L
'------------------------
MOVL C00186 BC00186 V=500.0
MOVL C00187 BC00187 V=166.7 PL=0
REFP 3 C00188 BC00188
CALL JOB:SEARCH-R1
SET P0360 P0006
SFTON P0360
MOVL C00189 BC00189 V=166.7 PL=0
REFP 3 C00190 BC00190
CALL JOB:SEARCH-R1
SET P0360 P0006
SFTON P0360
MOVL C00191 BC00191 V=166.7 PL=0
SFTOF
'------------------------
'W255A
'------------------------
MOVL C00192 BC00192 V=500.0
MOVL C00193 BC00193 V=166.7 PL=0
REFP 3 C00194 BC00194
CALL JOB:SEARCH-R1
SET P0361 P0006
SFTON P0361
MOVL C00195 BC00195 V=166.7 PL=0
REFP 3 C00196 BC00196
CALL JOB:SEARCH-R1
SET P0361 P0006
SFTON P0361
MOVL C00197 BC00197 V=166.7 PL=0
SFTOF
MOVL C00198 BC00198 V=666.7
MOVL C00199 BC00199 V=666.7
MOVL C00200 BC00200 V=666.7
MOVJ C00201 BC00201 VJ=40.00
MOVJ C00202 BC00202 VJ=40.00
MOVJ C00203 BC00203 VJ=40.00
COMM MOVJ C00204 BC00204 VJ=40.00
COMM MOVJ C00205 BC00205 VJ=40.00
COMM MOVJ C00206 BC00206 VJ=40.00
COMM MOVJ C00207 BC00207 VJ=40.00
COMM MOVJ C00208 BC00208 VJ=30.00
COMM '------------------------
COMM 'W61.3
COMM '------------------------
COMM MOVL C00209 BC00209 V=500.0
COMM MOVL C00210 BC00210 V=166.7 PL=0
COMM REFP 3 C00211 BC00211
COMM CALL JOB:SEARCH-R1
COMM SET P0400 P0006
COMM SFTON P0400
COMM MOVL C00212 BC00212 V=166.7 PL=0
COMM REFP 3 C00213 BC00213
COMM CALL JOB:SEARCH-R1
COMM SET P0400 P0006
COMM SFTON P0400
COMM MOVL C00214 BC00214 V=166.7 PL=0
COMM SFTOF
COMM 'BELKA PRZEJAZD
COMM MOVL C00215 BC00215 V=333.3
COMM '------------------------
COMM 'W61.5
COMM '------------------------
COMM MOVL C00216 BC00216 V=166.7 PL=0
COMM REFP 3 C00217 BC00217
COMM CALL JOB:SEARCH-R1
COMM SET P0401 P0006
COMM SFTON P0401
COMM MOVL C00218 BC00218 V=166.7 PL=0
COMM REFP 3 C00219 BC00219
COMM CALL JOB:SEARCH-R1
COMM SET P0401 P0006
COMM SFTON P0401
COMM MOVL C00220 BC00220 V=166.7 PL=0
COMM SFTOF
COMM '------------------------
COMM 'W61.7
COMM '------------------------
COMM MOVL C00221 BC00221 V=500.0
COMM MOVL C00222 BC00222 V=166.7 PL=0
COMM REFP 3 C00223 BC00223
COMM CALL JOB:SEARCH-R1
COMM SET P0402 P0006
COMM SFTON P0402
COMM MOVL C00224 BC00224 V=166.7 PL=0
COMM REFP 3 C00225 BC00225
COMM CALL JOB:SEARCH-R1
COMM SET P0402 P0006
COMM SFTON P0402
COMM MOVL C00226 BC00226 V=166.7 PL=0
COMM SFTOF
COMM MOVL C00227 BC00227 V=500.0
COMM '------------------------
COMM 'W61.10
COMM '------------------------
COMM MOVJ C00228 BC00228 VJ=30.00
COMM MOVJ C00229 BC00229 VJ=50.00
COMM MOVJ C00230 BC00230 VJ=50.00
COMM MOVL C00231 BC00231 V=500.0
COMM MOVL C00232 BC00232 V=166.7 PL=0
COMM REFP 3 C00233 BC00233
COMM CALL JOB:SEARCH-R1
COMM SET P0403 P0006
COMM SFTON P0403
COMM MOVL C00234 BC00234 V=166.7 PL=0
COMM REFP 3 C00235 BC00235
COMM CALL JOB:SEARCH-R1
COMM SET P0403 P0006
COMM SFTON P0403
COMM MOVL C00236 BC00236 V=166.7 PL=0
COMM SFTOF
COMM MOVL C00237 BC00237 V=333.3
COMM '------------------------
COMM 'W61.12
COMM '------------------------
COMM MOVL C00238 BC00238 V=666.7
COMM MOVL C00239 BC00239 V=166.7 PL=0
COMM REFP 3 C00240 BC00240
COMM CALL JOB:SEARCH-R1
COMM SET P0404 P0006
COMM SFTON P0404
COMM MOVL C00241 BC00241 V=166.7 PL=0
COMM REFP 3 C00242 BC00242
COMM CALL JOB:SEARCH-R1
COMM SET P0404 P0006
COMM SFTON P0404
COMM MOVL C00243 BC00243 V=166.7 PL=0
COMM SFTOF
COMM '------------------------
COMM 'W61.15
COMM '------------------------
COMM MOVL C00244 BC00244 V=666.7
COMM MOVL C00245 BC00245 V=166.7 PL=0
COMM REFP 3 C00246 BC00246
COMM CALL JOB:SEARCH-R1
COMM SET P0405 P0006
COMM SFTON P0405
COMM MOVL C00247 BC00247 V=166.7 PL=0
COMM REFP 3 C00248 BC00248
COMM CALL JOB:SEARCH-R1
COMM SET P0405 P0006
COMM SFTON P0405
COMM MOVL C00249 BC00249 V=166.7 PL=0
COMM SFTOF
COMM MOVL C00250 BC00250 V=666.7
COMM MOVJ C00251 BC00251 VJ=50.00
COMM MOVJ C00252 BC00252 VJ=50.00
COMM MOVJ C00253 BC00253 VJ=50.00
COMM '------------------------
COMM 'W61.17
COMM '------------------------
COMM MOVL C00254 BC00254 V=416.7
COMM MOVL C00255 BC00255 V=166.7 PL=0
COMM REFP 3 C00256 BC00256
COMM CALL JOB:SEARCH-R1
COMM SET P0406 P0006
COMM SFTON P0406
COMM MOVL C00257 BC00257 V=166.7 PL=0
COMM REFP 3 C00258 BC00258
COMM CALL JOB:SEARCH-R1
COMM SET P0406 P0006
COMM SFTON P0406
COMM MOVL C00259 BC00259 V=166.7 PL=0
COMM SFTOF
COMM MOVL C00260 BC00260 V=333.3
COMM '------------------------
COMM 'W61.20
COMM '------------------------
COMM MOVL C00261 BC00261 V=666.7
COMM MOVL C00262 BC00262 V=166.7 PL=0
COMM REFP 3 C00263 BC00263
COMM CALL JOB:SEARCH-R1
COMM SET P0407 P0006
COMM SFTON P0407
COMM MOVL C00264 BC00264 V=166.7 PL=0
COMM REFP 3 C00265 BC00265
COMM CALL JOB:SEARCH-R1
COMM SET P0407 P0006
COMM SFTON P0407
COMM MOVL C00266 BC00266 V=166.7 PL=0
COMM SFTOF
COMM '------------------------
COMM 'W61.23
COMM '------------------------
COMM MOVL C00267 BC00267 V=500.0
COMM MOVL C00268 BC00268 V=166.7 PL=0
COMM REFP 3 C00269 BC00269
COMM CALL JOB:SEARCH-R1
COMM SET P0408 P0006
COMM SFTON P0408
COMM MOVL C00270 BC00270 V=166.7 PL=0
COMM REFP 3 C00271 BC00271
COMM CALL JOB:SEARCH-R1
COMM SET P0408 P0006
COMM SFTON P0408
COMM MOVL C00272 BC00272 V=166.7 PL=0
COMM SFTOF
COMM MOVL C00273 BC00273 V=333.3
COMM MOVL C00274 BC00274 V=666.7
COMM MOVL C00275 BC00275 V=666.7
COMM '------------------------
COMM 'W61.25
COMM '------------------------
COMM MOVL C00276 BC00276 V=500.0
COMM MOVL C00277 BC00277 V=166.7 PL=0
COMM REFP 3 C00278 BC00278
COMM CALL JOB:SEARCH-R1
COMM SET P0409 P0006
COMM SFTON P0409
COMM MOVL C00279 BC00279 V=166.7 PL=0
COMM REFP 3 C00280 BC00280
COMM CALL JOB:SEARCH-R1
COMM SET P0409 P0006
COMM SFTON P0409
COMM MOVL C00281 BC00281 V=166.7 PL=0
COMM SFTOF
COMM MOVL C00282 BC00282 V=666.7
COMM MOVJ C00283 BC00283 VJ=50.00
COMM MOVJ C00284 BC00284 VJ=50.00
COMM GETE D040 P0409 (1)
COMM GETE D041 P0409 (2)
COMM GETE D042 P0409 (3)
COMM SETE P0410 (1) D040
COMM SETE P0410 (2) D041
COMM SETE P0410 (3) D042
COMM '------------------------
COMM 'W61.30
COMM '------------------------
COMM MOVL C00285 BC00285 V=500.0
COMM MOVL C00286 BC00286 V=166.7 PL=0
COMM REFP 3 C00287 BC00287
COMM CALL JOB:SEARCH-R1
COMM SET P0411 P0006
COMM SFTON P0411
COMM MOVL C00288 BC00288 V=166.7 PL=0
COMM REFP 3 C00289 BC00289
COMM CALL JOB:SEARCH-R1
COMM SET P0411 P0006
COMM SFTON P0411
COMM MOVL C00290 BC00290 V=166.7 PL=0
COMM SFTOF
COMM MOVL C00291 BC00291 V=666.7
COMM MOVJ C00292 BC00292 VJ=50.00
MOVJ C00293 BC00293 VJ=50.00
IFTHENEXP OT#(1457)=ON ANDEXP OT#(1441)=OFF
	 CALL JOB:TWIN_FRONT_SEARCH_-90ST-1_5340
ENDIF
IFTHENEXP OT#(1457)=OFF ANDEXP OT#(1441)=ON
	 CALL JOB:FRONT_SEARCH_-90ST-2_5340
ENDIF
MOVJ C00294 BC00294 VJ=60.00
MOVJ C00295 BC00295 VJ=50.00
MOVJ C00296 BC00296 VJ=50.00
MOVL C00297 BC00297 V=666.7
MOVJ C00298 BC00298 VJ=30.00
'------------------------
'W65.3
'------------------------
SFTON P0300
MOVL C00299 BC00299 V=333.3
MOVL C00300 BC00300 V=166.7 PL=0
MACRO1 MJ#(0) ARGF10
ARCON
MOVL C00301 BC00301 V=10.8
ARCOF
MOVL C00302 BC00302 V=166.7
SFTOF
'------------------------
'W65.5
'------------------------
SFTON P0301
MOVL C00303 BC00303 V=666.7
MOVL C00304 BC00304 V=166.7 PL=0
MACRO1 MJ#(0) ARGF9
ARCON
MOVL C00305 BC00305 V=8.3
ARCOF
MOVL C00306 BC00306 V=166.7
SFTOF
MOVL C00307 BC00307 V=500.0
MOVL C00308 BC00308 V=666.7
MOVJ C00309 BC00309 VJ=40.00
COMM MOVJ C00310 BC00310 VJ=60.00
COMM '::::::::::::::::::::::::::::::::
COMM '::::::::::::::::::::::::::::::::
COMM '::::::::::::::::::::::::::::::::
COMM '::::::::::::::::::::::::::::::::
COMM '::::::::::::::::::::::::::::::::
COMM MOVJ C00311 BC00311 VJ=50.00
COMM MOVJ C00312 BC00312 VJ=50.00
COMM MOVJ C00313 BC00313 VJ=40.00
COMM MOVJ C00314 BC00314 VJ=40.00
COMM MOVJ C00315 BC00315 VJ=40.00
COMM MOVJ C00316 BC00316 VJ=40.00
COMM MOVL C00317 BC00317 V=666.7
COMM '------------------------
COMM 'W61.3
COMM '------------------------
COMM SFTON P0400
COMM ARCOF
COMM MOVL C00318 BC00318 V=500.0
COMM SFTOF
COMM 'BELKA PRZEJAZD
COMM '------------------------
COMM 'W61.5
COMM '------------------------
COMM SFTON P0401
COMM MOVL C00319 BC00319 V=666.7
COMM MOVL C00320 BC00320 V=166.7 PL=0
COMM MACRO1 MJ#(0) ARGF24
COMM ARCON
COMM MOVL C00321 BC00321 V=7.5
COMM ARCOF
COMM MOVL C00322 BC00322 V=250.0
COMM SFTOF
COMM MOVL C00323 BC00323 V=500.0
COMM MOVJ C00324 BC00324 VJ=40.00
COMM MOVJ C00325 BC00325 VJ=40.00
COMM MOVJ C00326 BC00326 VJ=50.00
COMM MOVJ C00327 BC00327 VJ=50.00
MOVJ C00328 BC00328 VJ=50.00
MOVJ C00329 BC00329 VJ=50.00
MOVL C00330 BC00330 V=666.7
'------------------------
'W250A
'------------------------
SFTON P0354
MOVL C00331 BC00331 V=666.7
MOVL C00332 BC00332 V=166.7 PL=0
MACRO1 MJ#(0) ARGF9
ARCON
SFTOF
SFTON P0353
MOVL C00333 BC00333 V=11.7
ARCOF
MOVL C00334 BC00334 V=333.3
SFTOF
MOVJ C00335 BC00335 VJ=50.00
MOVJ C00336 BC00336 VJ=60.00
MOVJ C00337 BC00337 VJ=40.00
MOVJ C00338 BC00338 VJ=50.00
MOVJ C00339 BC00339 VJ=40.00
MOVJ C00340 BC00340 VJ=30.00
MOVJ C00341 BC00341 VJ=15.00
'------------------------
'W65.7
'------------------------
SFTON P0302
MOVL C00342 BC00342 V=833.3
MOVL C00343 BC00343 V=166.7 PL=0
MACRO1 MJ#(0) ARGF10
ARCON
MOVL C00344 BC00344 V=10.8
ARCOF
MOVL C00345 BC00345 V=166.7
SFTOF
'------------------------
'W65.10
'------------------------
SFTON P0303
MOVL C00346 BC00346 V=666.7
MOVL C00347 BC00347 V=166.7 PL=0
ARCON
MOVL C00348 BC00348 V=10.8
ARCOF
MOVL C00349 BC00349 V=166.7
SFTOF
MOVL C00350 BC00350 V=333.3
MOVL C00351 BC00351 V=666.7
MOVJ C00352 BC00352 VJ=30.00
MOVJ C00353 BC00353 VJ=30.00
MOVJ C00354 BC00354 VJ=30.00
MOVJ C00355 BC00355 VJ=50.00
COMM '::::::::::::::::::::::::::::::::
COMM '::::::::::::::::::::::::::::::::
COMM '------------------------
COMM 'W61.7
COMM '------------------------
COMM '::::::::::::::::::::::::::::::::
COMM '::::::::::::::::::::::::::::::::
COMM MOVJ C00356 BC00356 VJ=30.00
COMM MOVJ C00357 BC00357 VJ=30.00
COMM MOVJ C00358 BC00358 VJ=40.00
COMM SFTON P0402
COMM MOVL C00359 BC00359 V=500.0
COMM MOVL C00360 BC00360 V=166.7 PL=0
COMM MACRO1 MJ#(0) ARGF24
COMM ARCON
COMM MOVL C00361 BC00361 V=7.5
COMM ARCOF
COMM MOVL C00362 BC00362 V=250.0
COMM SFTOF
COMM MOVJ C00363 BC00363 VJ=30.00
COMM MOVJ C00364 BC00364 VJ=40.00
COMM MOVJ C00365 BC00365 VJ=50.00
COMM '------------------------
COMM 'W61.10
COMM '------------------------
COMM SFTON P0403
COMM MOVL C00366 BC00366 V=500.0
COMM MOVL C00367 BC00367 V=166.7 PL=0
COMM MACRO1 MJ#(0) ARGF24
COMM ARCON
COMM MOVL C00368 BC00368 V=7.5
COMM ARCOF
COMM MOVL C00369 BC00369 V=250.0
COMM SFTOF
COMM MOVL C00370 BC00370 V=500.0
COMM MOVL C00371 BC00371 V=666.7
COMM MOVL C00372 BC00372 V=666.7
COMM MOVJ C00373 BC00373 VJ=50.00
COMM MOVJ C00374 BC00374 VJ=50.00
COMM MOVJ C00375 BC00375 VJ=50.00
COMM '::::::::::::::::::::::::
COMM '::::::::::::::::::::::::
COMM '::::::::::::::::::::::::
COMM '::::::::::::::::::::::::
COMM '::::::::::::::::::::::::
COMM '::::::::::::::::::::::::
COMM '::::::::::::::::::::::::
MOVJ C00376 BC00376 VJ=50.00
MOVJ C00377 BC00377 VJ=50.00
MOVJ C00378 BC00378 VJ=50.00
'------------------------
'W251B
'------------------------
MOVL C00379 BC00379 V=500.0
MOVL C00380 BC00380 V=500.0
SFTON P0350
MOVL C00381 BC00381 V=166.7 PL=0
MACRO1 MJ#(0) ARGF9
ARCON
SFTOF
SFTON P0350
MOVL C00382 BC00382 V=11.3
SFTON P0349
MOVL C00383 BC00383 V=11.3
MOVL C00384 BC00384 V=11.3
ARCOF
MOVL C00385 BC00385 V=333.3
SFTOF
MOVJ C00386 BC00386 VJ=50.00
MOVJ C00387 BC00387 VJ=50.00
MOVJ C00388 BC00388 VJ=10.00
MOVJ C00389 BC00389 VJ=50.00
MOVJ C00390 BC00390 VJ=50.00
MOVJ C00391 BC00391 VJ=25.00
MOVJ C00392 BC00392 VJ=20.00
MOVJ C00393 BC00393 VJ=20.00
'------------------------
'W65.12
'------------------------
SFTON P0304
MOVL C00394 BC00394 V=333.3
MOVL C00395 BC00395 V=166.7 PL=0
MACRO1 MJ#(0) ARGF10
ARCON
MOVL C00396 BC00396 V=10.8
ARCOF
MOVL C00397 BC00397 V=166.7
SFTOF
'------------------------
'W65.15
'------------------------
SFTON P0305
MOVL C00398 BC00398 V=666.7
MOVL C00399 BC00399 V=166.7 PL=0
MACRO1 MJ#(0) ARGF9
ARCON
MOVL C00400 BC00400 V=10.8
ARCOF
MOVL C00401 BC00401 V=200.0
SFTOF
MOVL C00402 BC00402 V=250.0
MOVL C00403 BC00403 V=416.7
MOVL C00404 BC00404 V=666.7
COMM MOVJ C00405 BC00405 VJ=50.00
COMM MOVJ C00406 BC00406 VJ=50.00
COMM '::::::::::::::::::::::::
COMM '::::::::::::::::::::::::
COMM '::::::::::::::::::::::::
COMM '::::::::::::::::::::::::
COMM '::::::::::::::::::::::::
COMM '::::::::::::::::::::::::
COMM '::::::::::::::::::::::::
COMM MOVJ C00407 BC00407 VJ=50.00
COMM MOVJ C00408 BC00408 VJ=50.00
COMM MOVJ C00409 BC00409 VJ=50.00
COMM '::::::::::::::::::::::::::::::::
COMM '::::::::::::::::::::::::::::::::
COMM '------------------------
COMM 'W61.12
COMM '------------------------
COMM '::::::::::::::::::::::::::::::::
COMM '::::::::::::::::::::::::::::::::
COMM MOVL C00410 BC00410 V=833.3
COMM MOVL C00411 BC00411 V=666.7
COMM MOVL C00412 BC00412 V=500.0
COMM SFTON P0404
COMM MOVL C00413 BC00413 V=166.7 PL=0
COMM MACRO1 MJ#(0) ARGF24
COMM ARCON
COMM MOVL C00414 BC00414 V=6.7
COMM ARCOF
COMM MOVL C00415 BC00415 V=333.3
COMM SFTOF
COMM MOVL C00416 BC00416 V=500.0
COMM MOVL C00417 BC00417 V=666.7
COMM '------------------------
COMM 'W61.15
COMM '------------------------
COMM SFTON P0405
COMM MOVL C00418 BC00418 V=666.7
COMM MOVL C00419 BC00419 V=166.7 PL=0
COMM MACRO1 MJ#(0) ARGF24
COMM ARCON
COMM MOVL C00420 BC00420 V=6.7
COMM ARCOF
COMM MOVL C00421 BC00421 V=250.0
COMM SFTOF
COMM MOVJ C00422 BC00422 VJ=40.00
COMM MOVJ C00423 BC00423 VJ=40.00
COMM MOVJ C00424 BC00424 VJ=40.00
COMM MOVJ C00425 BC00425 VJ=40.00
COMM '::::::::::::::::::::::::
COMM '::::::::::::::::::::::::
COMM '::::::::::::::::::::::::
COMM '::::::::::::::::::::::::
COMM '::::::::::::::::::::::::
COMM '::::::::::::::::::::::::
COMM '::::::::::::::::::::::::
COMM MOVJ C00426 BC00426 VJ=40.00
COMM MOVJ C00427 BC00427 VJ=40.00
COMM '------------------------
COMM 'W252B
COMM '------------------------
SFTON P0359
MOVL C00428 BC00428 V=666.7
MOVL C00429 BC00429 V=166.7 PL=0
MACRO1 MJ#(0) ARGF9
ARCON
SFTOF
SFTON P0358
MOVL C00430 BC00430 V=10.8
ARCOF
MOVL C00431 BC00431 V=250.0
SFTOF
MOVJ C00432 BC00432 VJ=50.00
MOVJ C00433 BC00433 VJ=50.00
MOVJ C00434 BC00434 VJ=60.00
MOVJ C00435 BC00435 VJ=40.00
MOVJ C00436 BC00436 VJ=30.00
MOVL C00437 BC00437 V=500.0
MOVL C00438 BC00438 V=333.3
'------------------------
'W65.17
'------------------------
SFTON P0306
MOVL C00439 BC00439 V=333.3
MOVL C00440 BC00440 V=166.7 PL=0
MACRO1 MJ#(0) ARGF10
ARCON
MOVL C00441 BC00441 V=10.8
ARCOF
MOVL C00442 BC00442 V=166.7
SFTOF
MOVL C00443 BC00443 V=333.3
MOVL C00444 BC00444 V=500.0
MOVL C00445 BC00445 V=500.0
MOVJ C00446 BC00446 VJ=40.00
COMM MOVJ C00447 BC00447 VJ=60.00
COMM MOVJ C00448 BC00448 VJ=60.00
COMM '::::::::::::::::::::::::
COMM '::::::::::::::::::::::::
COMM '::::::::::::::::::::::::
COMM '::::::::::::::::::::::::
COMM '::::::::::::::::::::::::
COMM '::::::::::::::::::::::::
COMM '::::::::::::::::::::::::
COMM MOVJ C00449 BC00449 VJ=60.00
COMM '::::::::::::::::::::::::::::::::
COMM '::::::::::::::::::::::::::::::::
COMM '------------------------
COMM 'W61.17
COMM '------------------------
COMM '::::::::::::::::::::::::::::::::
COMM '::::::::::::::::::::::::::::::::
COMM SFTON P0406
COMM MOVJ C00450 BC00450 VJ=40.00
COMM MOVL C00451 BC00451 V=500.0
COMM MOVL C00452 BC00452 V=166.7 PL=0
COMM MACRO1 MJ#(0) ARGF24
COMM ARCON
COMM MOVL C00453 BC00453 V=6.7
COMM ARCOF
COMM MOVL C00454 BC00454 V=333.3
COMM SFTOF
COMM MOVJ C00455 BC00455 VJ=30.00
COMM MOVJ C00456 BC00456 VJ=40.00
COMM MOVJ C00457 BC00457 VJ=50.00
COMM '------------------------
COMM 'W253A
'------------------------
COMM MOVJ C00458 BC00458 VJ=50.00
MOVJ C00459 BC00459 VJ=50.00
SFTON P0356
MOVL C00460 BC00460 V=500.0
MOVL C00461 BC00461 V=500.0
MOVL C00462 BC00462 V=166.7 PL=0
MACRO1 MJ#(0) ARGF9
ARCON
SFTOF
SFTON P0355
MOVL C00463 BC00463 V=11.3
ARCOF
MOVL C00464 BC00464 V=333.3
SFTOF
MOVJ C00465 BC00465 VJ=50.00
MOVJ C00466 BC00466 VJ=50.00
MOVJ C00467 BC00467 VJ=50.00
MOVJ C00468 BC00468 VJ=50.00
MOVJ C00469 BC00469 VJ=50.00
MOVJ C00470 BC00470 VJ=50.00
MOVJ C00471 BC00471 VJ=40.00
MOVL C00472 BC00472 V=333.3
'------------------------
'W65.20
'------------------------
SFTON P0307
MOVL C00473 BC00473 V=500.0
MOVL C00474 BC00474 V=333.3
MOVL C00475 BC00475 V=166.7 PL=0
MACRO1 MJ#(0) ARGF10
ARCON
MOVL C00476 BC00476 V=10.8
ARCOF
MOVL C00477 BC00477 V=250.0
SFTOF
MOVL C00478 BC00478 V=666.7
MOVL C00479 BC00479 V=333.3
MOVL C00480 BC00480 V=500.0
MOVL C00481 BC00481 V=500.0
MOVJ C00482 BC00482 VJ=50.00
COMM MOVJ C00483 BC00483 VJ=50.00
COMM MOVJ C00484 BC00484 VJ=50.00
COMM MOVJ C00485 BC00485 VJ=50.00
COMM '::::::::::::::::::::::::
COMM '::::::::::::::::::::::::
COMM '::::::::::::::::::::::::
COMM '::::::::::::::::::::::::
COMM '::::::::::::::::::::::::
COMM '::::::::::::::::::::::::
COMM '::::::::::::::::::::::::
COMM MOVJ C00486 BC00486 VJ=40.00
COMM MOVJ C00487 BC00487 VJ=40.00
COMM '::::::::::::::::::::::::::::::::
COMM '::::::::::::::::::::::::::::::::
COMM '------------------------
COMM 'W61.20
COMM '------------------------
COMM '::::::::::::::::::::::::::::::::
COMM '::::::::::::::::::::::::::::::::
COMM SFTON P0407
COMM MOVL C00488 BC00488 V=666.7
COMM MOVL C00489 BC00489 V=333.3
COMM MOVL C00490 BC00490 V=166.7 PL=0
COMM MACRO1 MJ#(0) ARGF24
COMM ARCON
COMM MOVL C00491 BC00491 V=6.7
COMM ARCOF
COMM MOVL C00492 BC00492 V=250.0
COMM SFTOF
COMM '::::::::::::::::::::::::
COMM '::::::::::::::::::::::::
COMM '::::::::::::::::::::::::
COMM '::::::::::::::::::::::::
COMM '::::::::::::::::::::::::
COMM MOVL C00493 BC00493 V=500.0
COMM MOVJ C00494 BC00494 VJ=50.00
COMM MOVJ C00495 BC00495 VJ=50.00
COMM MOVJ C00496 BC00496 VJ=50.00
COMM '------------------------
COMM 'W254A
COMM '------------------------
COMM MOVJ C00497 BC00497 VJ=50.00
MOVJ C00498 BC00498 VJ=50.00
SFTON P0352
MOVL C00499 BC00499 V=666.7
MOVL C00500 BC00500 V=500.0
MOVL C00501 BC00501 V=250.0 PL=0
MACRO1 MJ#(0) ARGF9
ARCON
SFTOF
SFTON P0351
MOVL C00502 BC00502 V=11.2
ARCOF
MOVL C00503 BC00503 V=333.3
MOVL C00504 BC00504 V=666.7
SFTOF
COMM MOVJ C00505 BC00505 VJ=50.00
COMM MOVJ C00506 BC00506 VJ=80.00
COMM MOVJ C00507 BC00507 VJ=50.00
MOVJ C00508 BC00508 VJ=50.00
MOVJ C00509 BC00509 VJ=30.00
MOVJ C00510 BC00510 VJ=30.00
MOVJ C00511 BC00511 VJ=20.00
MOVL C00512 BC00512 V=666.7
'------------------------
'W65.23
'------------------------
SFTON P0308
MOVL C00513 BC00513 V=333.3
MOVL C00514 BC00514 V=166.7
MOVL C00515 BC00515 V=166.7 PL=0
MACRO1 MJ#(0) ARGF10
ARCON
MOVL C00516 BC00516 V=10.8
ARCOF
MOVL C00517 BC00517 V=250.0
SFTOF
'------------------------
'W65.25
'------------------------
SFTON P0309
MOVL C00518 BC00518 V=666.7
MOVL C00519 BC00519 V=166.7
MOVL C00520 BC00520 V=166.7 PL=0
ARCON
MOVL C00521 BC00521 V=10.8
ARCOF
MOVL C00522 BC00522 V=166.7
MOVL C00523 BC00523 V=166.7
SFTON P0310
MOVL C00524 BC00524 V=166.7
ARCON
MOVL C00525 BC00525 V=10.8
ARCOF
MOVL C00526 BC00526 V=250.0
MOVL C00527 BC00527 V=250.0
SFTOF
MOVL C00528 BC00528 V=250.0
MOVL C00529 BC00529 V=500.0
MOVL C00530 BC00530 V=666.7
MOVL C00531 BC00531 V=666.7
MOVJ C00532 BC00532 VJ=40.00
MOVJ C00533 BC00533 VJ=40.00
MOVJ C00534 BC00534 VJ=50.00
COMM '::::::::::::::::::::::::
COMM '::::::::::::::::::::::::
COMM '::::::::::::::::::::::::
COMM '::::::::::::::::::::::::
COMM '::::::::::::::::::::::::
COMM '::::::::::::::::::::::::
COMM '::::::::::::::::::::::::
COMM MOVJ C00535 BC00535 VJ=50.00
COMM MOVJ C00536 BC00536 VJ=50.00
COMM MOVJ C00537 BC00537 VJ=50.00
COMM '::::::::::::::::::::::::::::::::
COMM '::::::::::::::::::::::::::::::::
COMM '------------------------
COMM 'W61.23
COMM '------------------------
COMM '::::::::::::::::::::::::::::::::
COMM '::::::::::::::::::::::::::::::::
COMM SFTON P0408
COMM MOVL C00538 BC00538 V=500.0
COMM MOVL C00539 BC00539 V=666.7
COMM MOVL C00540 BC00540 V=166.7 PL=0
COMM MACRO1 MJ#(0) ARGF24
COMM ARCON
COMM MOVL C00541 BC00541 V=8.3
COMM ARCOF
COMM MOVL C00542 BC00542 V=250.0
COMM SFTOF
COMM MOVL C00543 BC00543 V=666.7
COMM '------------------------
COMM 'W61.25
COMM '------------------------
COMM SFTON P0409
COMM MOVL C00544 BC00544 V=500.0
COMM MOVL C00545 BC00545 V=166.7 PL=0
COMM MACRO1 MJ#(0) ARGF24
COMM ARCON
COMM MOVL C00546 BC00546 V=8.3
COMM ARCOF
COMM MOVL C00547 BC00547 V=166.7
COMM SFTOF
COMM MOVL C00548 BC00548 V=500.0
COMM MOVJ C00549 BC00549 VJ=20.00
COMM '::::::::::::::::::::::::
COMM '::::::::::::::::::::::::
COMM '::::::::::::::::::::::::
COMM '::::::::::::::::::::::::
COMM '::::::::::::::::::::::::
COMM MOVJ C00550 BC00550 VJ=50.00
COMM MOVJ C00551 BC00551 VJ=50.00
MOVJ C00552 BC00552 VJ=40.00
'------------------------
'W255A
MOVL C00553 BC00553 V=500.0
MOVL C00554 BC00554 V=666.7
SFTON P0361
MOVL C00555 BC00555 V=166.7 PL=0
MACRO1 MJ#(0) ARGF9
ARCON
MOVL C00556 BC00556 V=11.2
ARCOF
MOVL C00557 BC00557 V=333.3
SFTOF
MOVL C00558 BC00558 V=666.7
MOVL C00559 BC00559 V=666.7
MOVL C00560 BC00560 V=666.7
MOVJ C00561 BC00561 VJ=50.00
MOVJ C00562 BC00562 VJ=70.00
MOVJ C00563 BC00563 VJ=70.00
MOVJ C00564 BC00564 VJ=50.00
MOVJ C00565 BC00565 VJ=50.00
MOVJ C00566 BC00566 VJ=50.00
MOVL C00567 BC00567 V=500.0
'------------------------
'W31.28
'------------------------
MOVL C00568 BC00568 V=333.3
COMM MOVL C00569 BC00569 V=333.3
COMM MOVL C00570 BC00570 V=333.3
COMM MACRO1 MJ#(0) ARGF10
COMM MOVL C00571 BC00571 V=166.7
COMM ARCON
COMM MOVL C00572 BC00572 V=10.8
COMM ARCOF
COMM MOVL C00573 BC00573 V=200.0
COMM ARCON
COMM MOVL C00574 BC00574 V=10.8
COMM ARCOF
COMM MOVL C00575 BC00575 V=166.7
COMM SFTOF
COMM '------------------------
COMM 'W31.30
COMM '------------------------
SFTON P0311
MOVL C00576 BC00576 V=333.3
MOVL C00577 BC00577 V=166.7 PL=0
MACRO1 MJ#(0) ARGF9
ARCON
MOVL C00578 BC00578 V=10.8
ARCOF
MOVL C00579 BC00579 V=250.0
MOVL C00580 BC00580 V=333.3
SFTOF
SFTON P0312
MOVL C00581 BC00581 V=166.7
ARCON
MOVL C00582 BC00582 V=10.8
ARCOF
MOVL C00583 BC00583 V=166.7
ARCON
MOVL C00584 BC00584 V=10.8
ARCOF
SFTOF
MOVL C00585 BC00585 V=166.7
MOVL C00586 BC00586 V=500.0
MOVL C00587 BC00587 V=500.0
MOVL C00588 BC00588 V=666.7
MOVJ C00589 BC00589 VJ=25.00
COMM '::::::::::::::::::::::::
COMM '::::::::::::::::::::::::
COMM '::::::::::::::::::::::::
COMM '::::::::::::::::::::::::
COMM '::::::::::::::::::::::::
COMM '::::::::::::::::::::::::
COMM '::::::::::::::::::::::::
COMM MOVJ C00590 BC00590 VJ=20.00
COMM MOVJ C00591 BC00591 VJ=30.00
COMM '::::::::::::::::::::::::::::::::
COMM '::::::::::::::::::::::::::::::::
COMM '------------------------
COMM 'W61.30
COMM '------------------------
COMM '::::::::::::::::::::::::::::::::
COMM '::::::::::::::::::::::::::::::::
COMM SFTON P0411
COMM MOVL C00592 BC00592 V=500.0
COMM MOVL C00593 BC00593 V=166.7 PL=0
COMM MACRO1 MJ#(0) ARGF24
COMM ARCON
COMM MOVL C00594 BC00594 V=7.5
COMM ARCOF
COMM MOVL C00595 BC00595 V=250.0
COMM MOVL C00596 BC00596 V=500.0
COMM MOVL C00597 BC00597 V=166.7 PL=0
COMM MACRO1 MJ#(0) ARGF24
COMM ARCON
COMM MOVL C00598 BC00598 V=7.5
COMM ARCOF
COMM MOVL C00599 BC00599 V=250.0
COMM SFTOF
COMM MOVL C00600 BC00600 V=500.0
COMM SFTOF
COMM MOVL C00601 BC00601 V=500.0
COMM MOVJ C00602 BC00602 VJ=25.00
MOVJ C00603 BC00603 VJ=50.00
MOVJ C00604 BC00604 VJ=50.00
MOVJ C00605 BC00605 VJ=60.00
'------------------------
'W256A
'------------------------
MOVJ C00606 BC00606 VJ=60.00
MOVJ C00607 BC00607 VJ=60.00
SFTON P0358
MOVL C00608 BC00608 V=666.7
MOVL C00609 BC00609 V=250.0
MOVL C00610 BC00610 V=166.7 PL=0
MACRO1 MJ#(0) ARGF9
ARCON
SFTOF
SFTON P0357
MOVL C00611 BC00611 V=11.2
ARCOF
MOVL C00612 BC00612 V=333.3
SFTOF
MOVJ C00613 BC00613 VJ=50.00
MOVJ C00614 BC00614 VJ=50.00
IFTHENEXP OT#(1457)=ON ANDEXP OT#(1441)=OFF
	 CALL JOB:TWIN_FRONT_WELD_-90ST-2_5340
ENDIF
IFTHENEXP OT#(1457)=OFF ANDEXP OT#(1441)=ON
	 CALL JOB:FRONT_WELD_-90ST-2_5340
ENDIF
CALL JOB:MOVE_OUT_OF_TUNNEL
END
